LIN {X 0,Y 573.337,Z 321.881,A -85,B 0,C 180,E1 -2340.702,E2 -2340.702} C_VEL
LIN {X 0,Y 573.231,Z 321.897,A -85,B 0,C 180,E1 -2343.514,E2 -2343.514} C_VEL
LIN {X 0,Y 573.289,Z 321.888,A -85,B 0,C 180,E1 -2345.627,E2 -2345.627} C_VEL
LIN {X 0,Y 573.268,Z 321.89,A -85,B 0,C 180,E1 -2347.749,E2 -2347.749} C_VEL
LIN {X 0,Y 573.27,Z 321.892,A -85,B 0,C 180,E1 -2350.596,E2 -2350.596} C_VEL
LIN {X 0,Y 573.267,Z 321.891,A -85,B 0,C 180,E1 -2352.748,E2 -2352.748} C_VEL
LIN {X 0,Y 573.237,Z 321.894,A -85,B 0,C 180,E1 -2354.919,E2 -2354.919} C_VEL
LIN {X 0,Y 573.254,Z 321.892,A -85,B 0,C 180,E1 -2357.111,E2 -2357.111} C_VEL
LIN {X 0,Y 573.125,Z 322.237,A -85,B 0,C 180,E1 -2358.591,E2 -2358.591} C_VEL
LIN {X 0,Y 573.096,Z 326.558,A -85,B 0,C 180,E1 -2361.585,E2 -2361.585} C_VEL
LIN {X 0,Y 573.056,Z 329.759,A -85,B 0,C 180,E1 -2363.872,E2 -2363.872} C_VEL
LIN {X 0,Y 573.047,Z 330.361,A -85,B 0,C 180,E1 -2364.307,E2 -2364.307} C_VEL
LIN {X 0,Y 572.39,Z 331.226,A -85,B 0,C 180,E1 -2364.887,E2 -2364.887} C_VEL
LIN {X 0,Y 569.518,Z 332.787,A -85,B 0,C 180,E1 -2365.825,E2 -2365.825} C_VEL
LIN {X 0,Y 567.073,Z 334.053,A -85,B 0,C 180,E1 -2366.58,E2 -2366.58} C_VEL
LIN {X 0,Y 566.011,Z 334.964,A -85,B 0,C 180,E1 -2367.164,E2 -2367.164} C_VEL
LIN {X 0,Y 565.919,Z 335.251,A -85,B 0,C 180,E1 -2367.362,E2 -2367.362} C_VEL
LIN {X 0,Y 565.876,Z 338.726,A -85,B 0,C 180,E1 -2369.786,E2 -2369.786} C_VEL
LIN {X 0,Y 565.854,Z 342.602,A -85,B 0,C 180,E1 -2372.373,E2 -2372.373} C_VEL
LIN {X 0,Y 565.846,Z 346.578,A -85,B 0,C 180,E1 -2374.94,E2 -2374.94} C_VEL
LIN {X 0,Y 565.825,Z 350.574,A -85,B 0,C 180,E1 -2377.488,E2 -2377.488} C_VEL
LIN {X 0,Y 565.868,Z 354.863,A -85,B 0,C 180,E1 -2380.116,E2 -2380.116} C_VEL
LIN {X 0,Y 566.508,Z 362.319,A -85,B 0,C 180,E1 -2380.33,E2 -2380.33} C_VEL
LIN {X 0,Y 566.389,Z 373.209,A -85,B 0,C 180,E1 -2380.747,E2 -2380.747} C_VEL
LIN {X 0,Y 566.3,Z 382.804,A -85,B 0,C 180,E1 -2381.245,E2 -2381.245} C_VEL
LIN {X 0,Y 566.199,Z 390.332,A -85,B 0,C 180,E1 -2381.733,E2 -2381.733} C_VEL
LIN {X 0,Y 566.136,Z 397.915,A -85,B 0,C 180,E1 -2382.333,E2 -2382.333} C_VEL
LIN {X 0,Y 566.099,Z 405.454,A -85,B 0,C 180,E1 -2383.062,E2 -2383.062} C_VEL
LIN {X 0,Y 566.019,Z 413.662,A -85,B 0,C 180,E1 -2384.052,E2 -2384.052} C_VEL
LIN {X 0,Y 565.982,Z 419.96,A -85,B 0,C 180,E1 -2385.054,E2 -2385.054} C_VEL
LIN {X 0,Y 565.916,Z 424.329,A -85,B 0,C 180,E1 -2385.936,E2 -2385.936} C_VEL
LIN {X 0,Y 565.905,Z 426.671,A -85,B 0,C 180,E1 -2386.499,E2 -2386.499} C_VEL
LIN {X 0,Y 565.894,Z 428.668,A -85,B 0,C 180,E1 -2387.115,E2 -2387.115} C_VEL
LIN {X 0,Y 565.859,Z 431.271,A -85,B 0,C 180,E1 -2388.175,E2 -2388.175} C_VEL
LIN {X 0,Y 565.829,Z 432.675,A -85,B 0,C 180,E1 -2389.257,E2 -2389.257} C_VEL
LIN {X 0,Y 565.843,Z 432.888,A -85,B 0,C 180,E1 -2390.358,E2 -2390.358} C_VEL
LIN {X 0,Y 565.839,Z 431.745,A -85,B 0,C 180,E1 -2391.608,E2 -2391.608} C_VEL
LIN {X 0,Y 565.857,Z 429.634,A -85,B 0,C 180,E1 -2392.642,E2 -2392.642} C_VEL
LIN {X 0,Y 565.92,Z 425.738,A -85,B 0,C 180,E1 -2393.823,E2 -2393.823} C_VEL
LIN {X 0,Y 565.922,Z 421.824,A -85,B 0,C 180,E1 -2394.689,E2 -2394.689} C_VEL
LIN {X 0,Y 565.978,Z 416.587,A -85,B 0,C 180,E1 -2395.597,E2 -2395.597} C_VEL
LIN {X 0,Y 565.996,Z 411.667,A -85,B 0,C 180,E1 -2396.296,E2 -2396.296} C_VEL
LIN {X 0,Y 566.128,Z 404.978,A -85,B 0,C 180,E1 -2397.078,E2 -2397.078} C_VEL
LIN {X 0,Y 566.155,Z 398.125,A -85,B 0,C 180,E1 -2397.738,E2 -2397.738} C_VEL
LIN {X 0,Y 566.21,Z 390.149,A -85,B 0,C 180,E1 -2398.37,E2 -2398.37} C_VEL
LIN {X 0,Y 566.285,Z 380.733,A -85,B 0,C 180,E1 -2398.969,E2 -2398.969} C_VEL
LIN {X 0,Y 566.421,Z 370.239,A -85,B 0,C 180,E1 -2399.472,E2 -2399.472} C_VEL
LIN {X 0,Y 566.469,Z 359.574,A -85,B 0,C 180,E1 -2399.836,E2 -2399.836} C_VEL
LIN {X 0,Y 565.876,Z 354.723,A -85,B 0,C 180,E1 -2399.981,E2 -2399.981} C_VEL
LIN {X 0,Y 565.864,Z 350.509,A -85,B 0,C 180,E1 -2402.642,E2 -2402.642} C_VEL
LIN {X 0,Y 565.92,Z 346.759,A -85,B 0,C 180,E1 -2405.032,E2 -2405.032} C_VEL
LIN {X 0,Y 565.88,Z 341.975,A -85,B 0,C 180,E1 -2408.124,E2 -2408.124} C_VEL
LIN {X 0,Y 565.936,Z 337.526,A -85,B 0,C 180,E1 -2411.162,E2 -2411.162} C_VEL
LIN {X 0,Y 565.952,Z 334.388,A -85,B 0,C 180,E1 -2413.404,E2 -2413.404} C_VEL
LIN {X 0,Y 565.963,Z 330.08,A -85,B 0,C 180,E1 -2416.352,E2 -2416.352} C_VEL
LIN {X 0,Y 566.05,Z 325.919,A -85,B 0,C 180,E1 -2419.266,E2 -2419.266} C_VEL
LIN {X 0,Y 566.057,Z 322.872,A -85,B 0,C 180,E1 -2421.431,E2 -2421.431} C_VEL
LIN {X 0,Y 566.194,Z 322.774,A -85,B 0,C 180,E1 -2423.585,E2 -2423.585} C_VEL
LIN {X 0,Y 566.184,Z 322.773,A -85,B 0,C 180,E1 -2425.728,E2 -2425.728} C_VEL
LIN {X 0,Y 566.267,Z 322.762,A -85,B 0,C 180,E1 -2427.865,E2 -2427.865} C_VEL
LIN {X 0,Y 566.297,Z 322.761,A -85,B 0,C 180,E1 -2430.71,E2 -2430.71} C_VEL
LIN {X 0,Y 566.267,Z 322.762,A -85,B 0,C 180,E1 -2432.845,E2 -2432.845} C_VEL
LIN {X 0,Y 566.253,Z 322.767,A -85,B 0,C 180,E1 -2435.697,E2 -2435.697} C_VEL
LIN {X 0,Y 566.239,Z 322.765,A -85,B 0,C 180,E1 -2438.565,E2 -2438.565} C_VEL
LIN {X 0,Y 566.239,Z 322.766,A -85,B 0,C 180,E1 -2441.453,E2 -2441.453} C_VEL
LIN {X 0,Y 566.221,Z 322.767,A -85,B 0,C 180,E1 -2444.506,E2 -2444.506} C_VEL
LIN {X 0,Y 566.192,Z 322.771,A -85,B 0,C 180,E1 -2447.331,E2 -2447.331} C_VEL
LIN {X 0,Y 566.211,Z 322.771,A -85,B 0,C 180,E1 -2450.336,E2 -2450.336} C_VEL
LIN {X 0,Y 566.177,Z 322.773,A -85,B 0,C 180,E1 -2453.403,E2 -2453.403} C_VEL
LIN {X 0,Y 566.211,Z 322.769,A -85,B 0,C 180,E1 -2455.748,E2 -2455.748} C_VEL
LIN {X 0,Y 566.195,Z 322.77,A -85,B 0,C 180,E1 -2458.203,E2 -2458.203} C_VEL
LIN {X 0,Y 566.182,Z 322.772,A -85,B 0,C 180,E1 -2460.591,E2 -2460.591} C_VEL
LIN {X 0,Y 566.216,Z 322.768,A -85,B 0,C 180,E1 -2463.101,E2 -2463.101} C_VEL
LIN {X 0,Y 566.199,Z 322.771,A -85,B 0,C 180,E1 -2465.688,E2 -2465.688} C_VEL
LIN {X 0,Y 566.202,Z 322.773,A -85,B 0,C 180,E1 -2468.559,E2 -2468.559} C_VEL
LIN {X 0,Y 566.206,Z 322.771,A -85,B 0,C 180,E1 -2471.135,E2 -2471.135} C_VEL
LIN {X 0,Y 566.186,Z 322.771,A -85,B 0,C 180,E1 -2474.035,E2 -2474.035} C_VEL
LIN {X 0,Y 566.19,Z 322.774,A -85,B 0,C 180,E1 -2477.082,E2 -2477.082} C_VEL
LIN {X 0,Y 566.213,Z 322.768,A -85,B 0,C 180,E1 -2479.803,E2 -2479.803} C_VEL
LIN {X 0,Y 566.185,Z 322.772,A -85,B 0,C 180,E1 -2482.599,E2 -2482.599} C_VEL
LIN {X 0,Y 566.208,Z 322.77,A -85,B 0,C 180,E1 -2485.183,E2 -2485.183} C_VEL
LIN {X 0,Y 566.221,Z 322.77,A -85,B 0,C 180,E1 -2487.744,E2 -2487.744} C_VEL
LIN {X 0,Y 566.216,Z 322.771,A -85,B 0,C 180,E1 -2490.323,E2 -2490.323} C_VEL
LIN {X 0,Y 566.207,Z 322.772,A -85,B 0,C 180,E1 -2492.662,E2 -2492.662} C_VEL
LIN {X 0,Y 566.221,Z 322.77,A -85,B 0,C 180,E1 -2495.039,E2 -2495.039} C_VEL
LIN {X 0,Y 566.192,Z 322.773,A -85,B 0,C 180,E1 -2497.37,E2 -2497.37} C_VEL
LIN {X 0,Y 566.206,Z 322.769,A -85,B 0,C 180,E1 -2499.664,E2 -2499.664} C_VEL
LIN {X 0,Y 566.193,Z 322.772,A -85,B 0,C 180,E1 -2502.669,E2 -2502.669} C_VEL
LIN {X 0,Y 566.221,Z 322.767,A -85,B 0,C 180,E1 -2505.627,E2 -2505.627} C_VEL
LIN {X 0,Y 566.221,Z 322.769,A -85,B 0,C 180,E1 -2508.676,E2 -2508.676} C_VEL
LIN {X 0,Y 566.24,Z 322.765,A -85,B 0,C 180,E1 -2511.435,E2 -2511.435} C_VEL
LIN {X 0,Y 566.253,Z 322.765,A -85,B 0,C 180,E1 -2514.302,E2 -2514.302} C_VEL
LIN {X 0,Y 566.277,Z 322.761,A -85,B 0,C 180,E1 -2517.867,E2 -2517.867} C_VEL
LIN {X 0,Y 566.3,Z 322.76,A -85,B 0,C 180,E1 -2520.712,E2 -2520.712} C_VEL
LIN {X 0,Y 566.264,Z 322.763,A -85,B 0,C 180,E1 -2522.846,E2 -2522.846} C_VEL
LIN {X 0,Y 566.251,Z 322.766,A -85,B 0,C 180,E1 -2525.699,E2 -2525.699} C_VEL
LIN {X 0,Y 566.22,Z 322.767,A -85,B 0,C 180,E1 -2528.566,E2 -2528.566} C_VEL
LIN {X 0,Y 566.241,Z 322.767,A -85,B 0,C 180,E1 -2531.455,E2 -2531.455} C_VEL
LIN {X 0,Y 566.225,Z 322.766,A -85,B 0,C 180,E1 -2534.508,E2 -2534.508} C_VEL
LIN {X 0,Y 566.196,Z 322.771,A -85,B 0,C 180,E1 -2537.332,E2 -2537.332} C_VEL
LIN {X 0,Y 566.206,Z 322.77,A -85,B 0,C 180,E1 -2540.338,E2 -2540.338} C_VEL
LIN {X 0,Y 566.182,Z 322.773,A -85,B 0,C 180,E1 -2543.405,E2 -2543.405} C_VEL
LIN {X 0,Y 566.215,Z 322.769,A -85,B 0,C 180,E1 -2545.749,E2 -2545.749} C_VEL
LIN {X 0,Y 566.2,Z 322.77,A -85,B 0,C 180,E1 -2548.204,E2 -2548.204} C_VEL
LIN {X 0,Y 566.179,Z 322.772,A -85,B 0,C 180,E1 -2550.593,E2 -2550.593} C_VEL
LIN {X 0,Y 566.221,Z 322.768,A -85,B 0,C 180,E1 -2553.102,E2 -2553.102} C_VEL
LIN {X 0,Y 566.206,Z 322.771,A -85,B 0,C 180,E1 -2555.689,E2 -2555.689} C_VEL
LIN {X 0,Y 566.21,Z 322.77,A -85,B 0,C 180,E1 -2558.56,E2 -2558.56} C_VEL
LIN {X 0,Y 566.204,Z 322.77,A -85,B 0,C 180,E1 -2561.137,E2 -2561.137} C_VEL
LIN {X 0,Y 566.194,Z 322.771,A -85,B 0,C 180,E1 -2564.036,E2 -2564.036} C_VEL
LIN {X 0,Y 566.199,Z 322.771,A -85,B 0,C 180,E1 -2567.084,E2 -2567.084} C_VEL
LIN {X 0,Y 566.222,Z 322.767,A -85,B 0,C 180,E1 -2569.804,E2 -2569.804} C_VEL
LIN {X 0,Y 566.195,Z 322.771,A -85,B 0,C 180,E1 -2572.6,E2 -2572.6} C_VEL
LIN {X 0,Y 566.218,Z 322.771,A -85,B 0,C 180,E1 -2575.184,E2 -2575.184} C_VEL
LIN {X 0,Y 566.279,Z 322.886,A -85,B 0,C 180,E1 -2576.326,E2 -2576.326} C_VEL
LIN {X 0,Y 566.647,Z 327.07,A -85,B 0,C 180,E1 -2577.771,E2 -2577.771} C_VEL
LIN {X 0,Y 566.5,Z 334.622,A -85,B 0,C 180,E1 -2580.276,E2 -2580.276} C_VEL
LIN {X 0,Y 566.374,Z 343.367,A -85,B 0,C 180,E1 -2583.03,E2 -2583.03} C_VEL
LIN {X 0,Y 566.309,Z 351.29,A -85,B 0,C 180,E1 -2585.435,E2 -2585.435} C_VEL
LIN {X 0,Y 566.255,Z 360.365,A -85,B 0,C 180,E1 -2588.141,E2 -2588.141} C_VEL
LIN {X 0,Y 566.142,Z 370.65,A -85,B 0,C 180,E1 -2591.171,E2 -2591.171} C_VEL
LIN {X 0,Y 566.087,Z 379.591,A -85,B 0,C 180,E1 -2593.78,E2 -2593.78} C_VEL
LIN {X 0,Y 566.031,Z 388.533,A -85,B 0,C 180,E1 -2596.356,E2 -2596.356} C_VEL
LIN {X 0,Y 565.987,Z 397.114,A -85,B 0,C 180,E1 -2598.802,E2 -2598.802} C_VEL
LIN {X 0,Y 565.966,Z 401.306,A -85,B 0,C 180,E1 -2599.989,E2 -2599.989} C_VEL
LIN {X 0,Y 566.514,Z 408.45,A -85,B 0,C 180,E1 -2600.18,E2 -2600.18} C_VEL
LIN {X 0,Y 566.458,Z 416.916,A -85,B 0,C 180,E1 -2600.449,E2 -2600.449} C_VEL
LIN {X 0,Y 566.389,Z 425.418,A -85,B 0,C 180,E1 -2600.808,E2 -2600.808} C_VEL
LIN {X 0,Y 566.316,Z 433.746,A -85,B 0,C 180,E1 -2601.257,E2 -2601.257} C_VEL
LIN {X 0,Y 566.207,Z 441.783,A -85,B 0,C 180,E1 -2601.794,E2 -2601.794} C_VEL
LIN {X 0,Y 566.126,Z 450.442,A -85,B 0,C 180,E1 -2602.511,E2 -2602.511} C_VEL
LIN {X 0,Y 566.069,Z 459.353,A -85,B 0,C 180,E1 -2603.458,E2 -2603.458} C_VEL
LIN {X 0,Y 566.025,Z 465.618,A -85,B 0,C 180,E1 -2604.3,E2 -2604.3} C_VEL
LIN {X 0,Y 565.906,Z 469.993,A -85,B 0,C 180,E1 -2605.014,E2 -2605.014} C_VEL
LIN {X 0,Y 565.943,Z 475.152,A -85,B 0,C 180,E1 -2606.085,E2 -2606.085} C_VEL
LIN {X 0,Y 565.88,Z 478.938,A -85,B 0,C 180,E1 -2607.153,E2 -2607.153} C_VEL
LIN {X 0,Y 565.841,Z 480.684,A -85,B 0,C 180,E1 -2607.866,E2 -2607.866} C_VEL
LIN {X 0,Y 565.844,Z 481.935,A -85,B 0,C 180,E1 -2608.578,E2 -2608.578} C_VEL
LIN {X 0,Y 565.837,Z 482.71,A -85,B 0,C 180,E1 -2609.289,E2 -2609.289} C_VEL
LIN {X 0,Y 565.836,Z 483,A -85,B 0,C 180,E1 -2610.001,E2 -2610.001} C_VEL
LIN {X 0,Y 565.837,Z 482.709,A -85,B 0,C 180,E1 -2610.713,E2 -2610.713} C_VEL
LIN {X 0,Y 565.844,Z 481.933,A -85,B 0,C 180,E1 -2611.424,E2 -2611.424} C_VEL
LIN {X 0,Y 565.841,Z 480.679,A -85,B 0,C 180,E1 -2612.136,E2 -2612.136} C_VEL
LIN {X 0,Y 565.912,Z 477.785,A -85,B 0,C 180,E1 -2613.205,E2 -2613.205} C_VEL
LIN {X 0,Y 565.934,Z 475.144,A -85,B 0,C 180,E1 -2613.917,E2 -2613.917} C_VEL
LIN {X 0,Y 565.906,Z 469.981,A -85,B 0,C 180,E1 -2614.988,E2 -2614.988} C_VEL
LIN {X 0,Y 566.082,Z 463.179,A -85,B 0,C 180,E1 -2616.058,E2 -2616.058} C_VEL
LIN {X 0,Y 566.092,Z 456.174,A -85,B 0,C 180,E1 -2616.907,E2 -2616.907} C_VEL
LIN {X 0,Y 566.149,Z 448.395,A -85,B 0,C 180,E1 -2617.67,E2 -2617.67} C_VEL
LIN {X 0,Y 566.25,Z 440.531,A -85,B 0,C 180,E1 -2618.297,E2 -2618.297} C_VEL
LIN {X 0,Y 566.371,Z 430.715,A -85,B 0,C 180,E1 -2618.924,E2 -2618.924} C_VEL
LIN {X 0,Y 566.436,Z 419.281,A -85,B 0,C 180,E1 -2619.463,E2 -2619.463} C_VEL
LIN {X 0,Y 566.529,Z 409.215,A -85,B 0,C 180,E1 -2619.799,E2 -2619.799} C_VEL
LIN {X 0,Y 566.065,Z 402.339,A -85,B 0,C 180,E1 -2619.977,E2 -2619.977} C_VEL
LIN {X 0,Y 565.967,Z 401.299,A -85,B 0,C 180,E1 -2620.012,E2 -2620.012} C_VEL
LIN {X 0,Y 566.022,Z 392.358,A -85,B 0,C 180,E1 -2622.551,E2 -2622.551} C_VEL
LIN {X 0,Y 566.071,Z 382.139,A -85,B 0,C 180,E1 -2625.483,E2 -2625.483} C_VEL
LIN {X 0,Y 566.15,Z 371.921,A -85,B 0,C 180,E1 -2628.455,E2 -2628.455} C_VEL
LIN {X 0,Y 566.217,Z 362.937,A -85,B 0,C 180,E1 -2631.098,E2 -2631.098} C_VEL
LIN {X 0,Y 566.277,Z 353.823,A -85,B 0,C 180,E1 -2633.789,E2 -2633.789} C_VEL
LIN {X 0,Y 566.357,Z 344.685,A -85,B 0,C 180,E1 -2636.535,E2 -2636.535} C_VEL
LIN {X 0,Y 566.491,Z 335.795,A -85,B 0,C 180,E1 -2639.331,E2 -2639.331} C_VEL
LIN {X 0,Y 566.638,Z 328.27,A -85,B 0,C 180,E1 -2641.812,E2 -2641.812} C_VEL
LIN {X 0,Y 566.387,Z 323.621,A -85,B 0,C 180,E1 -2643.409,E2 -2643.409} C_VEL
LIN {X 0,Y 566.234,Z 322.768,A -85,B 0,C 180,E1 -2643.737,E2 -2643.737} C_VEL
LIN {X 0,Y 566.205,Z 322.77,A -85,B 0,C 180,E1 -2646.57,E2 -2646.57} C_VEL
LIN {X 0,Y 566.217,Z 322.77,A -85,B 0,C 180,E1 -2649.686,E2 -2649.686} C_VEL
LIN {X 0,Y 566.21,Z 322.774,A -85,B 0,C 180,E1 -2652.918,E2 -2652.918} C_VEL
LIN {X 0,Y 566.199,Z 322.772,A -85,B 0,C 180,E1 -2656.049,E2 -2656.049} C_VEL
LIN {X 0,Y 566.209,Z 322.769,A -85,B 0,C 180,E1 -2659.215,E2 -2659.215} C_VEL
LIN {X 0,Y 566.186,Z 322.772,A -85,B 0,C 180,E1 -2661.636,E2 -2661.636} C_VEL
LIN {X 0,Y 566.168,Z 322.775,A -85,B 0,C 180,E1 -2664.308,E2 -2664.308} C_VEL
LIN {X 0,Y 566.207,Z 322.771,A -85,B 0,C 180,E1 -2666.897,E2 -2666.897} C_VEL
LIN {X 0,Y 566.179,Z 322.776,A -85,B 0,C 180,E1 -2669.407,E2 -2669.407} C_VEL
LIN {X 0,Y 566.201,Z 322.773,A -85,B 0,C 180,E1 -2671.856,E2 -2671.856} C_VEL
LIN {X 0,Y 566.216,Z 322.77,A -85,B 0,C 180,E1 -2674.251,E2 -2674.251} C_VEL
LIN {X 0,Y 566.177,Z 322.774,A -85,B 0,C 180,E1 -2676.719,E2 -2676.719} C_VEL
LIN {X 0,Y 566.211,Z 322.769,A -85,B 0,C 180,E1 -2679.662,E2 -2679.662} C_VEL
LIN {X 0,Y 566.204,Z 322.77,A -85,B 0,C 180,E1 -2682.668,E2 -2682.668} C_VEL
LIN {X 0,Y 566.227,Z 322.768,A -85,B 0,C 180,E1 -2685.626,E2 -2685.626} C_VEL
LIN {X 0,Y 566.241,Z 322.765,A -85,B 0,C 180,E1 -2688.675,E2 -2688.675} C_VEL
LIN {X 0,Y 566.209,Z 322.77,A -85,B 0,C 180,E1 -2691.433,E2 -2691.433} C_VEL
LIN {X 0,Y 566.259,Z 322.765,A -85,B 0,C 180,E1 -2694.301,E2 -2694.301} C_VEL
LIN {X 0,Y 566.28,Z 322.762,A -85,B 0,C 180,E1 -2697.866,E2 -2697.866} C_VEL
LIN {X 0,Y 566.308,Z 322.757,A -85,B 0,C 180,E1 -2700.71,E2 -2700.71} C_VEL
LIN {X 0,Y 566.273,Z 322.761,A -85,B 0,C 180,E1 -2702.845,E2 -2702.845} C_VEL
LIN {X 0,Y 566.258,Z 322.764,A -85,B 0,C 180,E1 -2705.698,E2 -2705.698} C_VEL
LIN {X 0,Y 566.223,Z 322.767,A -85,B 0,C 180,E1 -2707.846,E2 -2707.846} C_VEL
LIN {X 0,Y 566.242,Z 322.768,A -85,B 0,C 180,E1 -2710.729,E2 -2710.729} C_VEL
LIN {X 0,Y 566.211,Z 322.771,A -85,B 0,C 180,E1 -2712.909,E2 -2712.909} C_VEL
LIN {X 0,Y 566.201,Z 322.772,A -85,B 0,C 180,E1 -2715.109,E2 -2715.109} C_VEL
LIN {X 0,Y 566.184,Z 322.773,A -85,B 0,C 180,E1 -2717.331,E2 -2717.331} C_VEL
LIN {X 0,Y 566.113,Z 322.784,A -85,B 0,C 180,E1 -2718.08,E2 -2718.08} C_VEL
LIN {X 0,Y 566.063,Z 323.28,A -85,B 0,C 180,E1 -2718.832,E2 -2718.832} C_VEL
LIN {X 0,Y 566.052,Z 326.899,A -85,B 0,C 180,E1 -2721.378,E2 -2721.378} C_VEL
LIN {X 0,Y 565.975,Z 330.828,A -85,B 0,C 180,E1 -2724.19,E2 -2724.19} C_VEL
LIN {X 0,Y 565.972,Z 334.186,A -85,B 0,C 180,E1 -2726.61,E2 -2726.61} C_VEL
LIN {X 0,Y 565.919,Z 335.251,A -85,B 0,C 180,E1 -2727.362,E2 -2727.362} C_VEL
LIN {X 0,Y 565.232,Z 336.148,A -85,B 0,C 180,E1 -2727.95,E2 -2727.95} C_VEL
LIN {X 0,Y 562.353,Z 337.767,A -85,B 0,C 180,E1 -2728.9,E2 -2728.9} C_VEL
LIN {X 0,Y 559.929,Z 339.082,A -85,B 0,C 180,E1 -2729.665,E2 -2729.665} C_VEL
LIN {X 0,Y 558.89,Z 340.031,A -85,B 0,C 180,E1 -2730.256,E2 -2730.256} C_VEL
LIN {X 0,Y 558.805,Z 340.331,A -85,B 0,C 180,E1 -2730.457,E2 -2730.457} C_VEL
LIN {X 0,Y 558.762,Z 343.568,A -85,B 0,C 180,E1 -2732.74,E2 -2732.74} C_VEL
LIN {X 0,Y 558.745,Z 347.513,A -85,B 0,C 180,E1 -2735.351,E2 -2735.351} C_VEL
LIN {X 0,Y 558.732,Z 351.698,A -85,B 0,C 180,E1 -2738.048,E2 -2738.048} C_VEL
LIN {X 0,Y 558.775,Z 354.79,A -85,B 0,C 180,E1 -2739.987,E2 -2739.987} C_VEL
LIN {X 0,Y 559.498,Z 361.692,A -85,B 0,C 180,E1 -2740.189,E2 -2740.189} C_VEL
LIN {X 0,Y 559.414,Z 372.799,A -85,B 0,C 180,E1 -2740.61,E2 -2740.61} C_VEL
LIN {X 0,Y 559.309,Z 381.698,A -85,B 0,C 180,E1 -2741.067,E2 -2741.067} C_VEL
LIN {X 0,Y 559.18,Z 389.687,A -85,B 0,C 180,E1 -2741.581,E2 -2741.581} C_VEL
LIN {X 0,Y 559.132,Z 396.739,A -85,B 0,C 180,E1 -2742.131,E2 -2742.131} C_VEL
LIN {X 0,Y 559.057,Z 404.361,A -85,B 0,C 180,E1 -2742.857,E2 -2742.857} C_VEL
LIN {X 0,Y 558.971,Z 410.72,A -85,B 0,C 180,E1 -2743.594,E2 -2743.594} C_VEL
LIN {X 0,Y 558.903,Z 415.222,A -85,B 0,C 180,E1 -2744.212,E2 -2744.212} C_VEL
LIN {X 0,Y 558.91,Z 420.013,A -85,B 0,C 180,E1 -2745,E2 -2745} C_VEL
LIN {X 0,Y 558.839,Z 423.945,A -85,B 0,C 180,E1 -2745.792,E2 -2745.792} C_VEL
LIN {X 0,Y 558.808,Z 427.909,A -85,B 0,C 180,E1 -2746.839,E2 -2746.839} C_VEL
LIN {X 0,Y 558.769,Z 430.737,A -85,B 0,C 180,E1 -2747.907,E2 -2747.907} C_VEL
LIN {X 0,Y 558.746,Z 432.616,A -85,B 0,C 180,E1 -2749.151,E2 -2749.151} C_VEL
LIN {X 0,Y 558.758,Z 432.993,A -85,B 0,C 180,E1 -2750.106,E2 -2750.106} C_VEL
LIN {X 0,Y 558.731,Z 432.251,A -85,B 0,C 180,E1 -2751.246,E2 -2751.246} C_VEL
LIN {X 0,Y 558.734,Z 431.251,A -85,B 0,C 180,E1 -2751.95,E2 -2751.95} C_VEL
LIN {X 0,Y 558.785,Z 429.141,A -85,B 0,C 180,E1 -2752.863,E2 -2752.863} C_VEL
LIN {X 0,Y 558.845,Z 426.176,A -85,B 0,C 180,E1 -2753.766,E2 -2753.766} C_VEL
LIN {X 0,Y 558.839,Z 421.404,A -85,B 0,C 180,E1 -2754.828,E2 -2754.828} C_VEL
LIN {X 0,Y 558.899,Z 417.435,A -85,B 0,C 180,E1 -2755.537,E2 -2755.537} C_VEL
LIN {X 0,Y 558.949,Z 411.399,A -85,B 0,C 180,E1 -2756.41,E2 -2756.41} C_VEL
LIN {X 0,Y 559.047,Z 404.951,A -85,B 0,C 180,E1 -2757.17,E2 -2757.17} C_VEL
LIN {X 0,Y 559.097,Z 398.37,A -85,B 0,C 180,E1 -2757.814,E2 -2757.814} C_VEL
LIN {X 0,Y 559.166,Z 390.358,A -85,B 0,C 180,E1 -2758.46,E2 -2758.46} C_VEL
LIN {X 0,Y 559.287,Z 380.547,A -85,B 0,C 180,E1 -2759.093,E2 -2759.093} C_VEL
LIN {X 0,Y 559.427,Z 369.369,A -85,B 0,C 180,E1 -2759.624,E2 -2759.624} C_VEL
LIN {X 0,Y 559.443,Z 359.915,A -85,B 0,C 180,E1 -2759.951,E2 -2759.951} C_VEL
LIN {X 0,Y 558.774,Z 354.712,A -85,B 0,C 180,E1 -2760.115,E2 -2760.115} C_VEL
LIN {X 0,Y 558.805,Z 349.825,A -85,B 0,C 180,E1 -2763.244,E2 -2763.244} C_VEL
LIN {X 0,Y 558.814,Z 346.373,A -85,B 0,C 180,E1 -2765.478,E2 -2765.478} C_VEL
LIN {X 0,Y 558.79,Z 342.847,A -85,B 0,C 180,E1 -2767.832,E2 -2767.832} C_VEL
LIN {X 0,Y 558.85,Z 338.459,A -85,B 0,C 180,E1 -2770.914,E2 -2770.914} C_VEL
LIN {X 0,Y 558.873,Z 335.274,A -85,B 0,C 180,E1 -2773.187,E2 -2773.187} C_VEL
LIN {X 0,Y 558.913,Z 330.916,A -85,B 0,C 180,E1 -2776.177,E2 -2776.177} C_VEL
LIN {X 0,Y 558.992,Z 326.76,A -85,B 0,C 180,E1 -2779.129,E2 -2779.129} C_VEL
LIN {X 0,Y 558.999,Z 323.698,A -85,B 0,C 180,E1 -2781.322,E2 -2781.322} C_VEL
LIN {X 0,Y 559.157,Z 323.65,A -85,B 0,C 180,E1 -2783.504,E2 -2783.504} C_VEL
LIN {X 0,Y 559.142,Z 323.65,A -85,B 0,C 180,E1 -2785.674,E2 -2785.674} C_VEL
LIN {X 0,Y 559.239,Z 323.637,A -85,B 0,C 180,E1 -2787.838,E2 -2787.838} C_VEL
LIN {X 0,Y 559.266,Z 323.637,A -85,B 0,C 180,E1 -2790.719,E2 -2790.719} C_VEL
LIN {X 0,Y 559.234,Z 323.638,A -85,B 0,C 180,E1 -2792.88,E2 -2792.88} C_VEL
LIN {X 0,Y 559.222,Z 323.642,A -85,B 0,C 180,E1 -2795.769,E2 -2795.769} C_VEL
LIN {X 0,Y 559.194,Z 323.642,A -85,B 0,C 180,E1 -2798.673,E2 -2798.673} C_VEL
LIN {X 0,Y 559.197,Z 323.644,A -85,B 0,C 180,E1 -2801.6,E2 -2801.6} C_VEL
LIN {X 0,Y 559.186,Z 323.643,A -85,B 0,C 180,E1 -2804.595,E2 -2804.595} C_VEL
LIN {X 0,Y 559.152,Z 323.649,A -85,B 0,C 180,E1 -2807.556,E2 -2807.556} C_VEL
LIN {X 0,Y 559.176,Z 323.645,A -85,B 0,C 180,E1 -2810.603,E2 -2810.603} C_VEL
LIN {X 0,Y 559.134,Z 323.652,A -85,B 0,C 180,E1 -2813.716,E2 -2813.716} C_VEL
LIN {X 0,Y 559.186,Z 323.645,A -85,B 0,C 180,E1 -2816.096,E2 -2816.096} C_VEL
LIN {X 0,Y 559.154,Z 323.649,A -85,B 0,C 180,E1 -2818.529,E2 -2818.529} C_VEL
LIN {X 0,Y 559.144,Z 323.652,A -85,B 0,C 180,E1 -2821.275,E2 -2821.275} C_VEL
LIN {X 0,Y 559.166,Z 323.646,A -85,B 0,C 180,E1 -2823.951,E2 -2823.951} C_VEL
LIN {X 0,Y 559.176,Z 323.645,A -85,B 0,C 180,E1 -2826.451,E2 -2826.451} C_VEL
LIN {X 0,Y 559.164,Z 323.647,A -85,B 0,C 180,E1 -2828.933,E2 -2828.933} C_VEL
LIN {X 0,Y 559.187,Z 323.644,A -85,B 0,C 180,E1 -2831.766,E2 -2831.766} C_VEL
LIN {X 0,Y 559.125,Z 323.653,A -85,B 0,C 180,E1 -2834.739,E2 -2834.739} C_VEL
LIN {X 0,Y 559.149,Z 323.649,A -85,B 0,C 180,E1 -2837.257,E2 -2837.257} C_VEL
LIN {X 0,Y 559.173,Z 323.645,A -85,B 0,C 180,E1 -2840.135,E2 -2840.135} C_VEL
LIN {X 0,Y 559.134,Z 323.653,A -85,B 0,C 180,E1 -2842.892,E2 -2842.892} C_VEL
LIN {X 0,Y 559.149,Z 323.651,A -85,B 0,C 180,E1 -2845.557,E2 -2845.557} C_VEL
LIN {X 0,Y 559.158,Z 323.649,A -85,B 0,C 180,E1 -2848.138,E2 -2848.138} C_VEL
LIN {X 0,Y 559.147,Z 323.65,A -85,B 0,C 180,E1 -2850.648,E2 -2850.648} C_VEL
LIN {X 0,Y 559.158,Z 323.647,A -85,B 0,C 180,E1 -2853.172,E2 -2853.172} C_VEL
LIN {X 0,Y 559.153,Z 323.648,A -85,B 0,C 180,E1 -2855.496,E2 -2855.496} C_VEL
LIN {X 0,Y 559.152,Z 323.649,A -85,B 0,C 180,E1 -2858.448,E2 -2858.448} C_VEL
LIN {X 0,Y 559.16,Z 323.648,A -85,B 0,C 180,E1 -2860.927,E2 -2860.927} C_VEL
LIN {X 0,Y 559.161,Z 323.648,A -85,B 0,C 180,E1 -2863.949,E2 -2863.949} C_VEL
LIN {X 0,Y 559.162,Z 323.65,A -85,B 0,C 180,E1 -2866.185,E2 -2866.185} C_VEL
LIN {X 0,Y 559.192,Z 323.645,A -85,B 0,C 180,E1 -2868.605,E2 -2868.605} C_VEL
LIN {X 0,Y 559.194,Z 323.643,A -85,B 0,C 180,E1 -2871.327,E2 -2871.327} C_VEL
LIN {X 0,Y 559.222,Z 323.64,A -85,B 0,C 180,E1 -2874.231,E2 -2874.231} C_VEL
LIN {X 0,Y 559.248,Z 323.637,A -85,B 0,C 180,E1 -2877.84,E2 -2877.84} C_VEL
LIN {X 0,Y 559.269,Z 323.636,A -85,B 0,C 180,E1 -2880.721,E2 -2880.721} C_VEL
LIN {X 0,Y 559.231,Z 323.64,A -85,B 0,C 180,E1 -2882.882,E2 -2882.882} C_VEL
LIN {X 0,Y 559.22,Z 323.641,A -85,B 0,C 180,E1 -2885.771,E2 -2885.771} C_VEL
LIN {X 0,Y 559.179,Z 323.644,A -85,B 0,C 180,E1 -2888.675,E2 -2888.675} C_VEL
LIN {X 0,Y 559.2,Z 323.646,A -85,B 0,C 180,E1 -2891.601,E2 -2891.601} C_VEL
LIN {X 0,Y 559.19,Z 323.642,A -85,B 0,C 180,E1 -2894.596,E2 -2894.596} C_VEL
LIN {X 0,Y 559.155,Z 323.65,A -85,B 0,C 180,E1 -2897.558,E2 -2897.558} C_VEL
LIN {X 0,Y 559.164,Z 323.648,A -85,B 0,C 180,E1 -2899.838,E2 -2899.838} C_VEL
LIN {X 0,Y 559.134,Z 323.651,A -85,B 0,C 180,E1 -2902.154,E2 -2902.154} C_VEL
LIN {X 0,Y 559.171,Z 323.647,A -85,B 0,C 180,E1 -2905.188,E2 -2905.188} C_VEL
LIN {X 0,Y 559.188,Z 323.644,A -85,B 0,C 180,E1 -2907.712,E2 -2907.712} C_VEL
LIN {X 0,Y 559.158,Z 323.647,A -85,B 0,C 180,E1 -2910.183,E2 -2910.183} C_VEL
LIN {X 0,Y 559.168,Z 323.646,A -85,B 0,C 180,E1 -2912.715,E2 -2912.715} C_VEL
LIN {X 0,Y 559.152,Z 323.648,A -85,B 0,C 180,E1 -2915.323,E2 -2915.323} C_VEL
LIN {X 0,Y 559.129,Z 323.652,A -85,B 0,C 180,E1 -2918.018,E2 -2918.018} C_VEL
LIN {X 0,Y 559.183,Z 323.645,A -85,B 0,C 180,E1 -2921.055,E2 -2921.055} C_VEL
LIN {X 0,Y 559.157,Z 323.647,A -85,B 0,C 180,E1 -2923.733,E2 -2923.733} C_VEL
LIN {X 0,Y 559.162,Z 323.65,A -85,B 0,C 180,E1 -2926.802,E2 -2926.802} C_VEL
LIN {X 0,Y 559.172,Z 323.649,A -85,B 0,C 180,E1 -2929.191,E2 -2929.191} C_VEL
LIN {X 0,Y 559.13,Z 323.651,A -85,B 0,C 180,E1 -2931.984,E2 -2931.984} C_VEL
LIN {X 0,Y 559.156,Z 323.648,A -85,B 0,C 180,E1 -2934.784,E2 -2934.784} C_VEL
LIN {X 0,Y 559.239,Z 323.815,A -85,B 0,C 180,E1 -2936.173,E2 -2936.173} C_VEL
LIN {X 0,Y 559.671,Z 328.303,A -85,B 0,C 180,E1 -2937.746,E2 -2937.746} C_VEL
LIN {X 0,Y 559.509,Z 335.246,A -85,B 0,C 180,E1 -2940.079,E2 -2940.079} C_VEL
LIN {X 0,Y 559.353,Z 343.397,A -85,B 0,C 180,E1 -2942.704,E2 -2942.704} C_VEL
LIN {X 0,Y 559.266,Z 351.32,A -85,B 0,C 180,E1 -2945.144,E2 -2945.144} C_VEL
LIN {X 0,Y 559.206,Z 360.268,A -85,B 0,C 180,E1 -2947.851,E2 -2947.851} C_VEL
LIN {X 0,Y 559.102,Z 369.19,A -85,B 0,C 180,E1 -2950.521,E2 -2950.521} C_VEL
LIN {X 0,Y 559.046,Z 378.314,A -85,B 0,C 180,E1 -2953.194,E2 -2953.194} C_VEL
LIN {X 0,Y 558.982,Z 388.533,A -85,B 0,C 180,E1 -2956.18,E2 -2956.18} C_VEL
LIN {X 0,Y 558.918,Z 398.751,A -85,B 0,C 180,E1 -2959.129,E2 -2959.129} C_VEL
LIN {X 0,Y 558.903,Z 401.306,A -85,B 0,C 180,E1 -2959.862,E2 -2959.862} C_VEL
LIN {X 0,Y 559.537,Z 408.449,A -85,B 0,C 180,E1 -2960.056,E2 -2960.056} C_VEL
LIN {X 0,Y 559.461,Z 416.914,A -85,B 0,C 180,E1 -2960.328,E2 -2960.328} C_VEL
LIN {X 0,Y 559.39,Z 425.415,A -85,B 0,C 180,E1 -2960.692,E2 -2960.692} C_VEL
LIN {X 0,Y 559.296,Z 433.744,A -85,B 0,C 180,E1 -2961.146,E2 -2961.146} C_VEL
LIN {X 0,Y 559.191,Z 441.78,A -85,B 0,C 180,E1 -2961.691,E2 -2961.691} C_VEL
LIN {X 0,Y 559.096,Z 450.443,A -85,B 0,C 180,E1 -2962.417,E2 -2962.417} C_VEL
LIN {X 0,Y 559.002,Z 458.957,A -85,B 0,C 180,E1 -2963.324,E2 -2963.324} C_VEL
LIN {X 0,Y 559.004,Z 464.441,A -85,B 0,C 180,E1 -2964.047,E2 -2964.047} C_VEL
LIN {X 0,Y 558.821,Z 469.994,A -85,B 0,C 180,E1 -2964.95,E2 -2964.95} C_VEL
LIN {X 0,Y 558.858,Z 475.153,A -85,B 0,C 180,E1 -2966.035,E2 -2966.035} C_VEL
LIN {X 0,Y 558.803,Z 478.939,A -85,B 0,C 180,E1 -2967.117,E2 -2967.117} C_VEL
LIN {X 0,Y 558.747,Z 480.685,A -85,B 0,C 180,E1 -2967.838,E2 -2967.838} C_VEL
LIN {X 0,Y 558.744,Z 481.934,A -85,B 0,C 180,E1 -2968.559,E2 -2968.559} C_VEL
LIN {X 0,Y 558.737,Z 482.709,A -85,B 0,C 180,E1 -2969.28,E2 -2969.28} C_VEL
LIN {X 0,Y 558.737,Z 483,A -85,B 0,C 180,E1 -2970.001,E2 -2970.001} C_VEL
LIN {X 0,Y 558.737,Z 482.708,A -85,B 0,C 180,E1 -2970.722,E2 -2970.722} C_VEL
LIN {X 0,Y 558.744,Z 481.931,A -85,B 0,C 180,E1 -2971.442,E2 -2971.442} C_VEL
LIN {X 0,Y 558.747,Z 480.68,A -85,B 0,C 180,E1 -2972.163,E2 -2972.163} C_VEL
LIN {X 0,Y 558.835,Z 477.784,A -85,B 0,C 180,E1 -2973.245,E2 -2973.245} C_VEL
LIN {X 0,Y 558.85,Z 475.145,A -85,B 0,C 180,E1 -2973.967,E2 -2973.967} C_VEL
LIN {X 0,Y 558.822,Z 469.981,A -85,B 0,C 180,E1 -2975.051,E2 -2975.051} C_VEL
LIN {X 0,Y 559.019,Z 463.178,A -85,B 0,C 180,E1 -2976.135,E2 -2976.135} C_VEL
LIN {X 0,Y 559.037,Z 455.736,A -85,B 0,C 180,E1 -2977.041,E2 -2977.041} C_VEL
LIN {X 0,Y 559.123,Z 448.393,A -85,B 0,C 180,E1 -2977.767,E2 -2977.767} C_VEL
LIN {X 0,Y 559.214,Z 440.529,A -85,B 0,C 180,E1 -2978.402,E2 -2978.402} C_VEL
LIN {X 0,Y 559.302,Z 432.213,A -85,B 0,C 180,E1 -2978.947,E2 -2978.947} C_VEL
LIN {X 0,Y 559.437,Z 421.593,A -85,B 0,C 180,E1 -2979.491,E2 -2979.491} C_VEL
LIN {X 0,Y 559.529,Z 410.046,A -85,B 0,C 180,E1 -2979.9,E2 -2979.9} C_VEL
LIN {X 0,Y 559.075,Z 402.986,A -85,B 0,C 180,E1 -2980.091,E2 -2980.091} C_VEL
LIN {X 0,Y 558.904,Z 401.299,A -85,B 0,C 180,E1 -2980.14,E2 -2980.14} C_VEL
LIN {X 0,Y 558.948,Z 392.358,A -85,B 0,C 180,E1 -2982.712,E2 -2982.712} C_VEL
LIN {X 0,Y 559.027,Z 382.139,A -85,B 0,C 180,E1 -2985.683,E2 -2985.683} C_VEL
LIN {X 0,Y 559.104,Z 371.888,A -85,B 0,C 180,E1 -2988.696,E2 -2988.696} C_VEL
LIN {X 0,Y 559.169,Z 362.185,A -85,B 0,C 180,E1 -2991.552,E2 -2991.552} C_VEL
LIN {X 0,Y 559.266,Z 352.386,A -85,B 0,C 180,E1 -2994.501,E2 -2994.501} C_VEL
LIN {X 0,Y 559.35,Z 343.242,A -85,B 0,C 180,E1 -2997.298,E2 -2997.298} C_VEL
LIN {X 0,Y 559.524,Z 334.465,A -85,B 0,C 180,E1 -3000.161,E2 -3000.161} C_VEL
LIN {X 0,Y 559.66,Z 328.224,A -85,B 0,C 180,E1 -3002.256,E2 -3002.256} C_VEL
LIN {X 0,Y 559.266,Z 324.005,A -85,B 0,C 180,E1 -3003.756,E2 -3003.756} C_VEL
LIN {X 0,Y 559.178,Z 323.647,A -85,B 0,C 180,E1 -3003.951,E2 -3003.951} C_VEL
LIN {X 0,Y 559.146,Z 323.652,A -85,B 0,C 180,E1 -3007.109,E2 -3007.109} C_VEL
LIN {X 0,Y 559.163,Z 323.648,A -85,B 0,C 180,E1 -3009.942,E2 -3009.942} C_VEL
LIN {X 0,Y 559.165,Z 323.65,A -85,B 0,C 180,E1 -3012.744,E2 -3012.744} C_VEL
LIN {X 0,Y 559.153,Z 323.649,A -85,B 0,C 180,E1 -3015.762,E2 -3015.762} C_VEL
LIN {X 0,Y 559.168,Z 323.646,A -85,B 0,C 180,E1 -3018.23,E2 -3018.23} C_VEL
LIN {X 0,Y 559.177,Z 323.648,A -85,B 0,C 180,E1 -3021.192,E2 -3021.192} C_VEL
LIN {X 0,Y 559.145,Z 323.65,A -85,B 0,C 180,E1 -3023.789,E2 -3023.789} C_VEL
LIN {X 0,Y 559.153,Z 323.648,A -85,B 0,C 180,E1 -3026.424,E2 -3026.424} C_VEL
LIN {X 0,Y 559.157,Z 323.648,A -85,B 0,C 180,E1 -3028.98,E2 -3028.98} C_VEL
LIN {X 0,Y 559.152,Z 323.65,A -85,B 0,C 180,E1 -3031.623,E2 -3031.623} C_VEL
LIN {X 0,Y 559.184,Z 323.646,A -85,B 0,C 180,E1 -3033.903,E2 -3033.903} C_VEL
LIN {X 0,Y 559.146,Z 323.651,A -85,B 0,C 180,E1 -3036.571,E2 -3036.571} C_VEL
LIN {X 0,Y 559.181,Z 323.644,A -85,B 0,C 180,E1 -3039.395,E2 -3039.395} C_VEL
LIN {X 0,Y 559.143,Z 323.649,A -85,B 0,C 180,E1 -3041.685,E2 -3041.685} C_VEL
LIN {X 0,Y 559.167,Z 323.647,A -85,B 0,C 180,E1 -3043.947,E2 -3043.947} C_VEL
LIN {X 0,Y 559.171,Z 323.647,A -85,B 0,C 180,E1 -3046.184,E2 -3046.184} C_VEL
LIN {X 0,Y 559.212,Z 323.641,A -85,B 0,C 180,E1 -3048.604,E2 -3048.604} C_VEL
LIN {X 0,Y 559.201,Z 323.643,A -85,B 0,C 180,E1 -3052.053,E2 -3052.053} C_VEL
LIN {X 0,Y 559.258,Z 323.635,A -85,B 0,C 180,E1 -3054.953,E2 -3054.953} C_VEL
LIN {X 0,Y 559.251,Z 323.637,A -85,B 0,C 180,E1 -3057.839,E2 -3057.839} C_VEL
LIN {X 0,Y 559.278,Z 323.632,A -85,B 0,C 180,E1 -3060.719,E2 -3060.719} C_VEL
LIN {X 0,Y 559.24,Z 323.637,A -85,B 0,C 180,E1 -3062.881,E2 -3062.881} C_VEL
LIN {X 0,Y 559.229,Z 323.64,A -85,B 0,C 180,E1 -3065.769,E2 -3065.769} C_VEL
LIN {X 0,Y 559.167,Z 323.647,A -85,B 0,C 180,E1 -3068.674,E2 -3068.674} C_VEL
LIN {X 0,Y 559.209,Z 323.642,A -85,B 0,C 180,E1 -3071.599,E2 -3071.599} C_VEL
LIN {X 0,Y 559.203,Z 323.643,A -85,B 0,C 180,E1 -3074.595,E2 -3074.595} C_VEL
LIN {X 0,Y 559.114,Z 323.655,A -85,B 0,C 180,E1 -3077.557,E2 -3077.557} C_VEL
LIN {X 0,Y 559.047,Z 323.665,A -85,B 0,C 180,E1 -3078.317,E2 -3078.317} C_VEL
LIN {X 0,Y 558.988,Z 324.857,A -85,B 0,C 180,E1 -3079.445,E2 -3079.445} C_VEL
LIN {X 0,Y 558.962,Z 328.665,A -85,B 0,C 180,E1 -3082.159,E2 -3082.159} C_VEL
LIN {X 0,Y 558.913,Z 332.73,A -85,B 0,C 180,E1 -3085.127,E2 -3085.127} C_VEL
LIN {X 0,Y 558.836,Z 336.373,A -85,B 0,C 180,E1 -3087.73,E2 -3087.73} C_VEL
LIN {X 0,Y 558.805,Z 340.331,A -85,B 0,C 180,E1 -3090.457,E2 -3090.457} C_VEL
LIN {X 0,Y 558.133,Z 341.262,A -85,B 0,C 180,E1 -3091.051,E2 -3091.051} C_VEL
LIN {X 0,Y 555.254,Z 342.861,A -85,B 0,C 180,E1 -3092.013,E2 -3092.013} C_VEL
LIN {X 0,Y 552.815,Z 344.147,A -85,B 0,C 180,E1 -3092.788,E2 -3092.788} C_VEL
LIN {X 0,Y 551.761,Z 345.07,A -85,B 0,C 180,E1 -3093.387,E2 -3093.387} C_VEL
LIN {X 0,Y 551.672,Z 345.362,A -85,B 0,C 180,E1 -3093.59,E2 -3093.59} C_VEL
LIN {X 0,Y 551.662,Z 348.608,A -85,B 0,C 180,E1 -3095.874,E2 -3095.874} C_VEL
LIN {X 0,Y 551.639,Z 353.405,A -85,B 0,C 180,E1 -3098.999,E2 -3098.999} C_VEL
LIN {X 0,Y 551.671,Z 354.715,A -85,B 0,C 180,E1 -3099.846,E2 -3099.846} C_VEL
LIN {X 0,Y 552.52,Z 363.25,A -85,B 0,C 180,E1 -3100.112,E2 -3100.112} C_VEL
LIN {X 0,Y 552.396,Z 373.304,A -85,B 0,C 180,E1 -3100.514,E2 -3100.514} C_VEL
LIN {X 0,Y 552.267,Z 382.592,A -85,B 0,C 180,E1 -3101.007,E2 -3101.007} C_VEL
LIN {X 0,Y 552.119,Z 390.95,A -85,B 0,C 180,E1 -3101.566,E2 -3101.566} C_VEL
LIN {X 0,Y 552.049,Z 398.306,A -85,B 0,C 180,E1 -3102.171,E2 -3102.171} C_VEL
LIN {X 0,Y 551.981,Z 405.929,A -85,B 0,C 180,E1 -3102.934,E2 -3102.934} C_VEL
LIN {X 0,Y 551.898,Z 412.13,A -85,B 0,C 180,E1 -3103.694,E2 -3103.694} C_VEL
LIN {X 0,Y 551.817,Z 418.881,A -85,B 0,C 180,E1 -3104.72,E2 -3104.72} C_VEL
LIN {X 0,Y 551.76,Z 424.131,A -85,B 0,C 180,E1 -3105.782,E2 -3105.782} C_VEL
LIN {X 0,Y 551.735,Z 427.147,A -85,B 0,C 180,E1 -3106.556,E2 -3106.556} C_VEL
LIN {X 0,Y 551.684,Z 430.191,A -85,B 0,C 180,E1 -3107.634,E2 -3107.634} C_VEL
LIN {X 0,Y 551.662,Z 432.123,A -85,B 0,C 180,E1 -3108.731,E2 -3108.731} C_VEL
LIN {X 0,Y 551.642,Z 432.942,A -85,B 0,C 180,E1 -3109.853,E2 -3109.853} C_VEL
LIN {X 0,Y 551.637,Z 432.575,A -85,B 0,C 180,E1 -3110.999,E2 -3110.999} C_VEL
LIN {X 0,Y 551.662,Z 430.537,A -85,B 0,C 180,E1 -3112.301,E2 -3112.301} C_VEL
LIN {X 0,Y 551.705,Z 428.134,A -85,B 0,C 180,E1 -3113.221,E2 -3113.221} C_VEL
LIN {X 0,Y 551.737,Z 424.871,A -85,B 0,C 180,E1 -3114.129,E2 -3114.129} C_VEL
LIN {X 0,Y 551.765,Z 420.684,A -85,B 0,C 180,E1 -3115.027,E2 -3115.027} C_VEL
LIN {X 0,Y 551.802,Z 415.467,A -85,B 0,C 180,E1 -3115.916,E2 -3115.916} C_VEL
LIN {X 0,Y 551.932,Z 409.002,A -85,B 0,C 180,E1 -3116.801,E2 -3116.801} C_VEL
LIN {X 0,Y 552.036,Z 399.811,A -85,B 0,C 180,E1 -3117.783,E2 -3117.783} C_VEL
LIN {X 0,Y 552.122,Z 392.01,A -85,B 0,C 180,E1 -3118.444,E2 -3118.444} C_VEL
LIN {X 0,Y 552.199,Z 384.426,A -85,B 0,C 180,E1 -3118.971,E2 -3118.971} C_VEL
LIN {X 0,Y 552.289,Z 376.876,A -85,B 0,C 180,E1 -3119.401,E2 -3119.401} C_VEL
LIN {X 0,Y 552.431,Z 368.847,A -85,B 0,C 180,E1 -3119.767,E2 -3119.767} C_VEL
LIN {X 0,Y 552.431,Z 360.438,A -85,B 0,C 180,E1 -3120.063,E2 -3120.063} C_VEL
LIN {X 0,Y 551.681,Z 354.709,A -85,B 0,C 180,E1 -3120.248,E2 -3120.248} C_VEL
LIN {X 0,Y 551.7,Z 350.331,A -85,B 0,C 180,E1 -3123.087,E2 -3123.087} C_VEL
LIN {X 0,Y 551.713,Z 346.084,A -85,B 0,C 180,E1 -3125.943,E2 -3125.943} C_VEL
LIN {X 0,Y 551.715,Z 342.542,A -85,B 0,C 180,E1 -3128.417,E2 -3128.417} C_VEL
LIN {X 0,Y 551.788,Z 339.391,A -85,B 0,C 180,E1 -3130.66,E2 -3130.66} C_VEL
LIN {X 0,Y 551.809,Z 336.11,A -85,B 0,C 180,E1 -3132.965,E2 -3132.965} C_VEL
LIN {X 0,Y 551.828,Z 331.763,A -85,B 0,C 180,E1 -3135.996,E2 -3135.996} C_VEL
LIN {X 0,Y 551.941,Z 327.593,A -85,B 0,C 180,E1 -3138.988,E2 -3138.988} C_VEL
LIN {X 0,Y 551.95,Z 324.548,A -85,B 0,C 180,E1 -3141.21,E2 -3141.21} C_VEL
LIN {X 0,Y 552.124,Z 324.525,A -85,B 0,C 180,E1 -3143.421,E2 -3143.421} C_VEL
LIN {X 0,Y 552.222,Z 324.513,A -85,B 0,C 180,E1 -3144.888,E2 -3144.888} C_VEL
LIN {X 0,Y 552.211,Z 324.513,A -85,B 0,C 180,E1 -3147.811,E2 -3147.811} C_VEL
LIN {X 0,Y 552.236,Z 324.512,A -85,B 0,C 180,E1 -3150.728,E2 -3150.728} C_VEL
LIN {X 0,Y 552.2,Z 324.515,A -85,B 0,C 180,E1 -3152.917,E2 -3152.917} C_VEL
LIN {X 0,Y 552.192,Z 324.517,A -85,B 0,C 180,E1 -3155.843,E2 -3155.843} C_VEL
LIN {X 0,Y 552.162,Z 324.518,A -85,B 0,C 180,E1 -3158.785,E2 -3158.785} C_VEL
LIN {X 0,Y 552.153,Z 324.523,A -85,B 0,C 180,E1 -3161.75,E2 -3161.75} C_VEL
LIN {X 0,Y 552.124,Z 324.523,A -85,B 0,C 180,E1 -3164.748,E2 -3164.748} C_VEL
LIN {X 0,Y 552.103,Z 324.529,A -85,B 0,C 180,E1 -3167.788,E2 -3167.788} C_VEL
LIN {X 0,Y 552.123,Z 324.526,A -85,B 0,C 180,E1 -3170.1,E2 -3170.1} C_VEL
LIN {X 0,Y 552.084,Z 324.53,A -85,B 0,C 180,E1 -3172.45,E2 -3172.45} C_VEL
LIN {X 0,Y 552.143,Z 324.523,A -85,B 0,C 180,E1 -3175.35,E2 -3175.35} C_VEL
LIN {X 0,Y 552.114,Z 324.524,A -85,B 0,C 180,E1 -3178.097,E2 -3178.097} C_VEL
LIN {X 0,Y 552.102,Z 324.526,A -85,B 0,C 180,E1 -3180.608,E2 -3180.608} C_VEL
LIN {X 0,Y 552.116,Z 324.525,A -85,B 0,C 180,E1 -3183.184,E2 -3183.184} C_VEL
LIN {X 0,Y 552.1,Z 324.528,A -85,B 0,C 180,E1 -3185.841,E2 -3185.841} C_VEL
LIN {X 0,Y 552.112,Z 324.525,A -85,B 0,C 180,E1 -3189.062,E2 -3189.062} C_VEL
LIN {X 0,Y 552.157,Z 324.519,A -85,B 0,C 180,E1 -3191.441,E2 -3191.441} C_VEL
LIN {X 0,Y 552.081,Z 324.531,A -85,B 0,C 180,E1 -3194.532,E2 -3194.532} C_VEL
LIN {X 0,Y 552.115,Z 324.524,A -85,B 0,C 180,E1 -3197.584,E2 -3197.584} C_VEL
LIN {X 0,Y 552.121,Z 324.525,A -85,B 0,C 180,E1 -3200.474,E2 -3200.474} C_VEL
LIN {X 0,Y 552.108,Z 324.526,A -85,B 0,C 180,E1 -3203.315,E2 -3203.315} C_VEL
LIN {X 0,Y 552.127,Z 324.523,A -85,B 0,C 180,E1 -3205.94,E2 -3205.94} C_VEL
LIN {X 0,Y 552.103,Z 324.526,A -85,B 0,C 180,E1 -3208.541,E2 -3208.541} C_VEL
LIN {X 0,Y 552.114,Z 324.527,A -85,B 0,C 180,E1 -3211.437,E2 -3211.437} C_VEL
LIN {X 0,Y 552.116,Z 324.525,A -85,B 0,C 180,E1 -3214.356,E2 -3214.356} C_VEL
LIN {X 0,Y 552.128,Z 324.523,A -85,B 0,C 180,E1 -3216.76,E2 -3216.76} C_VEL
LIN {X 0,Y 552.114,Z 324.525,A -85,B 0,C 180,E1 -3219.121,E2 -3219.121} C_VEL
LIN {X 0,Y 552.12,Z 324.525,A -85,B 0,C 180,E1 -3221.445,E2 -3221.445} C_VEL
LIN {X 0,Y 552.11,Z 324.528,A -85,B 0,C 180,E1 -3223.738,E2 -3223.738} C_VEL
LIN {X 0,Y 552.124,Z 324.526,A -85,B 0,C 180,E1 -3226.005,E2 -3226.005} C_VEL
LIN {X 0,Y 552.149,Z 324.52,A -85,B 0,C 180,E1 -3228.994,E2 -3228.994} C_VEL
LIN {X 0,Y 552.153,Z 324.521,A -85,B 0,C 180,E1 -3231.952,E2 -3231.952} C_VEL
LIN {X 0,Y 552.222,Z 324.512,A -85,B 0,C 180,E1 -3234.89,E2 -3234.89} C_VEL
LIN {X 0,Y 552.219,Z 324.512,A -85,B 0,C 180,E1 -3237.813,E2 -3237.813} C_VEL
LIN {X 0,Y 552.239,Z 324.511,A -85,B 0,C 180,E1 -3240.73,E2 -3240.73} C_VEL
LIN {X 0,Y 552.198,Z 324.516,A -85,B 0,C 180,E1 -3242.919,E2 -3242.919} C_VEL
LIN {X 0,Y 552.19,Z 324.516,A -85,B 0,C 180,E1 -3245.845,E2 -3245.845} C_VEL
LIN {X 0,Y 552.15,Z 324.52,A -85,B 0,C 180,E1 -3248.786,E2 -3248.786} C_VEL
LIN {X 0,Y 552.155,Z 324.522,A -85,B 0,C 180,E1 -3251.751,E2 -3251.751} C_VEL
LIN {X 0,Y 552.127,Z 324.522,A -85,B 0,C 180,E1 -3254.749,E2 -3254.749} C_VEL
LIN {X 0,Y 552.106,Z 324.528,A -85,B 0,C 180,E1 -3257.789,E2 -3257.789} C_VEL
LIN {X 0,Y 552.122,Z 324.526,A -85,B 0,C 180,E1 -3260.102,E2 -3260.102} C_VEL
LIN {X 0,Y 552.088,Z 324.53,A -85,B 0,C 180,E1 -3262.452,E2 -3262.452} C_VEL
LIN {X 0,Y 552.148,Z 324.521,A -85,B 0,C 180,E1 -3265.352,E2 -3265.352} C_VEL
LIN {X 0,Y 552.12,Z 324.524,A -85,B 0,C 180,E1 -3268.098,E2 -3268.098} C_VEL
LIN {X 0,Y 552.102,Z 324.526,A -85,B 0,C 180,E1 -3270.61,E2 -3270.61} C_VEL
LIN {X 0,Y 552.122,Z 324.525,A -85,B 0,C 180,E1 -3273.186,E2 -3273.186} C_VEL
LIN {X 0,Y 552.107,Z 324.528,A -85,B 0,C 180,E1 -3275.842,E2 -3275.842} C_VEL
LIN {X 0,Y 552.119,Z 324.525,A -85,B 0,C 180,E1 -3279.063,E2 -3279.063} C_VEL
LIN {X 0,Y 552.133,Z 324.522,A -85,B 0,C 180,E1 -3281.445,E2 -3281.445} C_VEL
LIN {X 0,Y 552.091,Z 324.53,A -85,B 0,C 180,E1 -3284.533,E2 -3284.533} C_VEL
LIN {X 0,Y 552.125,Z 324.523,A -85,B 0,C 180,E1 -3287.586,E2 -3287.586} C_VEL
LIN {X 0,Y 552.129,Z 324.526,A -85,B 0,C 180,E1 -3290.474,E2 -3290.474} C_VEL
LIN {X 0,Y 552.111,Z 324.525,A -85,B 0,C 180,E1 -3293.317,E2 -3293.317} C_VEL
LIN {X 0,Y 552.196,Z 324.546,A -85,B 0,C 180,E1 -3295.945,E2 -3295.945} C_VEL
LIN {X 0,Y 552.709,Z 329.53,A -85,B 0,C 180,E1 -3297.722,E2 -3297.722} C_VEL
LIN {X 0,Y 552.483,Z 338.253,A -85,B 0,C 180,E1 -3300.677,E2 -3300.677} C_VEL
LIN {X 0,Y 552.351,Z 345.288,A -85,B 0,C 180,E1 -3302.957,E2 -3302.957} C_VEL
LIN {X 0,Y 552.241,Z 353.689,A -85,B 0,C 180,E1 -3305.57,E2 -3305.57} C_VEL
LIN {X 0,Y 552.124,Z 362.686,A -85,B 0,C 180,E1 -3308.339,E2 -3308.339} C_VEL
LIN {X 0,Y 552.041,Z 371.667,A -85,B 0,C 180,E1 -3311.057,E2 -3311.057} C_VEL
LIN {X 0,Y 551.957,Z 380.847,A -85,B 0,C 180,E1 -3313.734,E2 -3313.734} C_VEL
LIN {X 0,Y 551.905,Z 389.81,A -85,B 0,C 180,E1 -3316.375,E2 -3316.375} C_VEL
LIN {X 0,Y 551.855,Z 398.751,A -85,B 0,C 180,E1 -3318.988,E2 -3318.988} C_VEL
LIN {X 0,Y 551.839,Z 401.306,A -85,B 0,C 180,E1 -3319.73,E2 -3319.73} C_VEL
LIN {X 0,Y 552.544,Z 410.111,A -85,B 0,C 180,E1 -3319.975,E2 -3319.975} C_VEL
LIN {X 0,Y 552.435,Z 421.632,A -85,B 0,C 180,E1 -3320.389,E2 -3320.389} C_VEL
LIN {X 0,Y 552.274,Z 432.241,A -85,B 0,C 180,E1 -3320.94,E2 -3320.94} C_VEL
LIN {X 0,Y 552.189,Z 440.549,A -85,B 0,C 180,E1 -3321.492,E2 -3321.492} C_VEL
LIN {X 0,Y 552.076,Z 448.407,A -85,B 0,C 180,E1 -3322.135,E2 -3322.135} C_VEL
LIN {X 0,Y 551.99,Z 455.92,A -85,B 0,C 180,E1 -3322.888,E2 -3322.888} C_VEL
LIN {X 0,Y 551.956,Z 463.431,A -85,B 0,C 180,E1 -3323.82,E2 -3323.82} C_VEL
LIN {X 0,Y 551.743,Z 469.994,A -85,B 0,C 180,E1 -3324.885,E2 -3324.885} C_VEL
LIN {X 0,Y 551.778,Z 475.153,A -85,B 0,C 180,E1 -3325.984,E2 -3325.984} C_VEL
LIN {X 0,Y 551.729,Z 478.939,A -85,B 0,C 180,E1 -3327.08,E2 -3327.08} C_VEL
LIN {X 0,Y 551.657,Z 480.684,A -85,B 0,C 180,E1 -3327.811,E2 -3327.811} C_VEL
LIN {X 0,Y 551.644,Z 481.933,A -85,B 0,C 180,E1 -3328.541,E2 -3328.541} C_VEL
LIN {X 0,Y 551.638,Z 482.708,A -85,B 0,C 180,E1 -3329.271,E2 -3329.271} C_VEL
LIN {X 0,Y 551.637,Z 483,A -85,B 0,C 180,E1 -3330.001,E2 -3330.001} C_VEL
LIN {X 0,Y 551.638,Z 482.707,A -85,B 0,C 180,E1 -3330.731,E2 -3330.731} C_VEL
LIN {X 0,Y 551.644,Z 481.93,A -85,B 0,C 180,E1 -3331.461,E2 -3331.461} C_VEL
LIN {X 0,Y 551.658,Z 480.679,A -85,B 0,C 180,E1 -3332.191,E2 -3332.191} C_VEL
LIN {X 0,Y 551.76,Z 477.784,A -85,B 0,C 180,E1 -3333.287,E2 -3333.287} C_VEL
LIN {X 0,Y 551.772,Z 475.145,A -85,B 0,C 180,E1 -3334.018,E2 -3334.018} C_VEL
LIN {X 0,Y 551.743,Z 469.981,A -85,B 0,C 180,E1 -3335.116,E2 -3335.116} C_VEL
LIN {X 0,Y 551.957,Z 463.398,A -85,B 0,C 180,E1 -3336.184,E2 -3336.184} C_VEL
LIN {X 0,Y 551.995,Z 455.735,A -85,B 0,C 180,E1 -3337.132,E2 -3337.132} C_VEL
LIN {X 0,Y 552.078,Z 448.391,A -85,B 0,C 180,E1 -3337.866,E2 -3337.866} C_VEL
LIN {X 0,Y 552.19,Z 440.526,A -85,B 0,C 180,E1 -3338.509,E2 -3338.509} C_VEL
LIN {X 0,Y 552.279,Z 432.211,A -85,B 0,C 180,E1 -3339.061,E2 -3339.061} C_VEL
LIN {X 0,Y 552.449,Z 421.592,A -85,B 0,C 180,E1 -3339.613,E2 -3339.613} C_VEL
LIN {X 0,Y 552.559,Z 410.045,A -85,B 0,C 180,E1 -3340.027,E2 -3340.027} C_VEL
LIN {X 0,Y 552.017,Z 402.985,A -85,B 0,C 180,E1 -3340.222,E2 -3340.222} C_VEL
LIN {X 0,Y 551.839,Z 401.299,A -85,B 0,C 180,E1 -3340.272,E2 -3340.272} C_VEL
LIN {X 0,Y 551.86,Z 391.081,A -85,B 0,C 180,E1 -3343.253,E2 -3343.253} C_VEL
LIN {X 0,Y 551.95,Z 382.139,A -85,B 0,C 180,E1 -3345.889,E2 -3345.889} C_VEL
LIN {X 0,Y 552.022,Z 372.931,A -85,B 0,C 180,E1 -3348.56,E2 -3348.56} C_VEL
LIN {X 0,Y 552.096,Z 363.838,A -85,B 0,C 180,E1 -3351.273,E2 -3351.273} C_VEL
LIN {X 0,Y 552.228,Z 353.544,A -85,B 0,C 180,E1 -3354.433,E2 -3354.433} C_VEL
LIN {X 0,Y 552.307,Z 345.151,A -85,B 0,C 180,E1 -3357.034,E2 -3357.034} C_VEL
LIN {X 0,Y 552.488,Z 336.89,A -85,B 0,C 180,E1 -3359.743,E2 -3359.743} C_VEL
LIN {X 0,Y 552.68,Z 329.421,A -85,B 0,C 180,E1 -3362.282,E2 -3362.282} C_VEL
LIN {X 0,Y 552.343,Z 325.755,A -85,B 0,C 180,E1 -3363.608,E2 -3363.608} C_VEL
LIN {X 0,Y 552.137,Z 324.525,A -85,B 0,C 180,E1 -3364.104,E2 -3364.104} C_VEL
LIN {X 0,Y 552.111,Z 324.527,A -85,B 0,C 180,E1 -3366.747,E2 -3366.747} C_VEL
LIN {X 0,Y 552.132,Z 324.526,A -85,B 0,C 180,E1 -3369.528,E2 -3369.528} C_VEL
LIN {X 0,Y 552.136,Z 324.524,A -85,B 0,C 180,E1 -3372.426,E2 -3372.426} C_VEL
LIN {X 0,Y 552.097,Z 324.529,A -85,B 0,C 180,E1 -3375.562,E2 -3375.562} C_VEL
LIN {X 0,Y 552.126,Z 324.525,A -85,B 0,C 180,E1 -3378.554,E2 -3378.554} C_VEL
LIN {X 0,Y 552.12,Z 324.525,A -85,B 0,C 180,E1 -3381.411,E2 -3381.411} C_VEL
LIN {X 0,Y 552.091,Z 324.528,A -85,B 0,C 180,E1 -3384.156,E2 -3384.156} C_VEL
LIN {X 0,Y 552.112,Z 324.526,A -85,B 0,C 180,E1 -3386.814,E2 -3386.814} C_VEL
LIN {X 0,Y 552.104,Z 324.529,A -85,B 0,C 180,E1 -3389.39,E2 -3389.39} C_VEL
LIN {X 0,Y 552.099,Z 324.529,A -85,B 0,C 180,E1 -3391.901,E2 -3391.901} C_VEL
LIN {X 0,Y 552.162,Z 324.519,A -85,B 0,C 180,E1 -3394.65,E2 -3394.65} C_VEL
LIN {X 0,Y 552.098,Z 324.529,A -85,B 0,C 180,E1 -3397.549,E2 -3397.549} C_VEL
LIN {X 0,Y 552.151,Z 324.521,A -85,B 0,C 180,E1 -3400.375,E2 -3400.375} C_VEL
LIN {X 0,Y 552.14,Z 324.521,A -85,B 0,C 180,E1 -3402.976,E2 -3402.976} C_VEL
LIN {X 0,Y 552.137,Z 324.524,A -85,B 0,C 180,E1 -3406.004,E2 -3406.004} C_VEL
LIN {X 0,Y 552.167,Z 324.518,A -85,B 0,C 180,E1 -3408.993,E2 -3408.993} C_VEL
LIN {X 0,Y 552.155,Z 324.522,A -85,B 0,C 180,E1 -3411.951,E2 -3411.951} C_VEL
LIN {X 0,Y 552.232,Z 324.51,A -85,B 0,C 180,E1 -3414.888,E2 -3414.888} C_VEL
LIN {X 0,Y 552.223,Z 324.513,A -85,B 0,C 180,E1 -3417.811,E2 -3417.811} C_VEL
LIN {X 0,Y 552.248,Z 324.508,A -85,B 0,C 180,E1 -3420.728,E2 -3420.728} C_VEL
LIN {X 0,Y 552.207,Z 324.513,A -85,B 0,C 180,E1 -3422.917,E2 -3422.917} C_VEL
LIN {X 0,Y 552.2,Z 324.516,A -85,B 0,C 180,E1 -3425.843,E2 -3425.843} C_VEL
LIN {X 0,Y 552.14,Z 324.522,A -85,B 0,C 180,E1 -3428.785,E2 -3428.785} C_VEL
LIN {X 0,Y 552.166,Z 324.521,A -85,B 0,C 180,E1 -3431.75,E2 -3431.75} C_VEL
LIN {X 0,Y 552.14,Z 324.523,A -85,B 0,C 180,E1 -3434.747,E2 -3434.747} C_VEL
LIN {X 0,Y 552.106,Z 324.527,A -85,B 0,C 180,E1 -3437.309,E2 -3437.309} C_VEL
LIN {X 0,Y 551.959,Z 324.547,A -85,B 0,C 180,E1 -3438.56,E2 -3438.56} C_VEL
LIN {X 0,Y 551.895,Z 327.551,A -85,B 0,C 180,E1 -3440.888,E2 -3440.888} C_VEL
LIN {X 0,Y 551.87,Z 331.232,A -85,B 0,C 180,E1 -3443.52,E2 -3443.52} C_VEL
LIN {X 0,Y 551.824,Z 335.269,A -85,B 0,C 180,E1 -3446.471,E2 -3446.471} C_VEL
LIN {X 0,Y 551.75,Z 338.772,A -85,B 0,C 180,E1 -3448.948,E2 -3448.948} C_VEL
LIN {X 0,Y 551.721,Z 342.428,A -85,B 0,C 180,E1 -3451.483,E2 -3451.483} C_VEL
LIN {X 0,Y 551.672,Z 345.362,A -85,B 0,C 180,E1 -3453.59,E2 -3453.59} C_VEL
LIN {X 0,Y 550.987,Z 346.267,A -85,B 0,C 180,E1 -3454.193,E2 -3454.193} C_VEL
LIN {X 0,Y 548.097,Z 347.879,A -85,B 0,C 180,E1 -3455.168,E2 -3455.168} C_VEL
LIN {X 0,Y 545.669,Z 349.182,A -85,B 0,C 180,E1 -3455.953,E2 -3455.953} C_VEL
LIN {X 0,Y 544.639,Z 350.125,A -85,B 0,C 180,E1 -3456.56,E2 -3456.56} C_VEL
LIN {X 0,Y 544.561,Z 350.424,A -85,B 0,C 180,E1 -3456.766,E2 -3456.766} C_VEL
LIN {X 0,Y 544.58,Z 354.723,A -85,B 0,C 180,E1 -3459.717,E2 -3459.717} C_VEL
LIN {X 0,Y 545.537,Z 363.115,A -85,B 0,C 180,E1 -3459.979,E2 -3459.979} C_VEL
LIN {X 0,Y 545.369,Z 374.402,A -85,B 0,C 180,E1 -3460.445,E2 -3460.445} C_VEL
LIN {X 0,Y 545.25,Z 383.341,A -85,B 0,C 180,E1 -3460.936,E2 -3460.936} C_VEL
LIN {X 0,Y 545.079,Z 391.829,A -85,B 0,C 180,E1 -3461.523,E2 -3461.523} C_VEL
LIN {X 0,Y 544.988,Z 400.313,A -85,B 0,C 180,E1 -3462.251,E2 -3462.251} C_VEL
LIN {X 0,Y 544.874,Z 408.42,A -85,B 0,C 180,E1 -3463.125,E2 -3463.125} C_VEL
LIN {X 0,Y 544.783,Z 414.375,A -85,B 0,C 180,E1 -3463.926,E2 -3463.926} C_VEL
LIN {X 0,Y 544.732,Z 419.644,A -85,B 0,C 180,E1 -3464.797,E2 -3464.797} C_VEL
LIN {X 0,Y 544.683,Z 424.56,A -85,B 0,C 180,E1 -3465.832,E2 -3465.832} C_VEL
LIN {X 0,Y 544.641,Z 426.343,A -85,B 0,C 180,E1 -3466.269,E2 -3466.269} C_VEL
LIN {X 0,Y 544.616,Z 429.644,A -85,B 0,C 180,E1 -3467.352,E2 -3467.352} C_VEL
LIN {X 0,Y 544.593,Z 431.789,A -85,B 0,C 180,E1 -3468.458,E2 -3468.458} C_VEL
LIN {X 0,Y 544.545,Z 432.925,A -85,B 0,C 180,E1 -3469.81,E2 -3469.81} C_VEL
LIN {X 0,Y 544.548,Z 432.712,A -85,B 0,C 180,E1 -3470.772,E2 -3470.772} C_VEL
LIN {X 0,Y 544.536,Z 431.378,A -85,B 0,C 180,E1 -3471.931,E2 -3471.931} C_VEL
LIN {X 0,Y 544.614,Z 428.528,A -85,B 0,C 180,E1 -3473.136,E2 -3473.136} C_VEL
LIN {X 0,Y 544.658,Z 425.581,A -85,B 0,C 180,E1 -3474.009,E2 -3474.009} C_VEL
LIN {X 0,Y 544.695,Z 421.374,A -85,B 0,C 180,E1 -3474.958,E2 -3474.958} C_VEL
LIN {X 0,Y 544.749,Z 416.571,A -85,B 0,C 180,E1 -3475.817,E2 -3475.817} C_VEL
LIN {X 0,Y 544.833,Z 410.705,A -85,B 0,C 180,E1 -3476.666,E2 -3476.666} C_VEL
LIN {X 0,Y 544.933,Z 404.345,A -85,B 0,C 180,E1 -3477.421,E2 -3477.421} C_VEL
LIN {X 0,Y 545.029,Z 397.629,A -85,B 0,C 180,E1 -3478.083,E2 -3478.083} C_VEL
LIN {X 0,Y 545.109,Z 389.439,A -85,B 0,C 180,E1 -3478.748,E2 -3478.748} C_VEL
LIN {X 0,Y 545.293,Z 379.951,A -85,B 0,C 180,E1 -3479.363,E2 -3479.363} C_VEL
LIN {X 0,Y 545.435,Z 369.028,A -85,B 0,C 180,E1 -3479.886,E2 -3479.886} C_VEL
LIN {X 0,Y 545.422,Z 360.976,A -85,B 0,C 180,E1 -3480.178,E2 -3480.178} C_VEL
LIN {X 0,Y 544.61,Z 354.709,A -85,B 0,C 180,E1 -3480.382,E2 -3480.382} C_VEL
LIN {X 0,Y 544.609,Z 350.611,A -85,B 0,C 180,E1 -3483.149,E2 -3483.149} C_VEL
LIN {X 0,Y 544.626,Z 347.052,A -85,B 0,C 180,E1 -3485.61,E2 -3485.61} C_VEL
LIN {X 0,Y 544.64,Z 343.257,A -85,B 0,C 180,E1 -3488.289,E2 -3488.289} C_VEL
LIN {X 0,Y 544.686,Z 339.221,A -85,B 0,C 180,E1 -3491.181,E2 -3491.181} C_VEL
LIN {X 0,Y 544.723,Z 335.918,A -85,B 0,C 180,E1 -3493.509,E2 -3493.509} C_VEL
LIN {X 0,Y 544.749,Z 332.659,A -85,B 0,C 180,E1 -3495.81,E2 -3495.81} C_VEL
LIN {X 0,Y 544.896,Z 328.467,A -85,B 0,C 180,E1 -3498.844,E2 -3498.844} C_VEL
LIN {X 0,Y 544.889,Z 325.428,A -85,B 0,C 180,E1 -3501.095,E2 -3501.095} C_VEL
LIN {X 0,Y 545.091,Z 325.401,A -85,B 0,C 180,E1 -3503.336,E2 -3503.336} C_VEL
LIN {X 0,Y 545.197,Z 325.388,A -85,B 0,C 180,E1 -3504.822,E2 -3504.822} C_VEL
LIN {X 0,Y 545.183,Z 325.388,A -85,B 0,C 180,E1 -3507.783,E2 -3507.783} C_VEL
LIN {X 0,Y 545.206,Z 325.388,A -85,B 0,C 180,E1 -3510.738,E2 -3510.738} C_VEL
LIN {X 0,Y 545.166,Z 325.391,A -85,B 0,C 180,E1 -3512.955,E2 -3512.955} C_VEL
LIN {X 0,Y 545.163,Z 325.392,A -85,B 0,C 180,E1 -3515.919,E2 -3515.919} C_VEL
LIN {X 0,Y 545.118,Z 325.396,A -85,B 0,C 180,E1 -3518.899,E2 -3518.899} C_VEL
LIN {X 0,Y 545.124,Z 325.397,A -85,B 0,C 180,E1 -3521.903,E2 -3521.903} C_VEL
LIN {X 0,Y 545.073,Z 325.401,A -85,B 0,C 180,E1 -3524.943,E2 -3524.943} C_VEL
LIN {X 0,Y 545.071,Z 325.403,A -85,B 0,C 180,E1 -3528.025,E2 -3528.025} C_VEL
LIN {X 0,Y 545.088,Z 325.402,A -85,B 0,C 180,E1 -3530.371,E2 -3530.371} C_VEL
LIN {X 0,Y 545.078,Z 325.402,A -85,B 0,C 180,E1 -3533.558,E2 -3533.558} C_VEL
LIN {X 0,Y 545.075,Z 325.402,A -85,B 0,C 180,E1 -3535.999,E2 -3535.999} C_VEL
LIN {X 0,Y 545.08,Z 325.403,A -85,B 0,C 180,E1 -3538.749,E2 -3538.749} C_VEL
LIN {X 0,Y 545.064,Z 325.403,A -85,B 0,C 180,E1 -3541.682,E2 -3541.682} C_VEL
LIN {X 0,Y 545.072,Z 325.402,A -85,B 0,C 180,E1 -3544.562,E2 -3544.562} C_VEL
LIN {X 0,Y 545.055,Z 325.407,A -85,B 0,C 180,E1 -3547.301,E2 -3547.301} C_VEL
LIN {X 0,Y 545.08,Z 325.4,A -85,B 0,C 180,E1 -3550.14,E2 -3550.14} C_VEL
LIN {X 0,Y 545.053,Z 325.404,A -85,B 0,C 180,E1 -3552.697,E2 -3552.697} C_VEL
LIN {X 0,Y 545.048,Z 325.405,A -85,B 0,C 180,E1 -3555.167,E2 -3555.167} C_VEL
LIN {X 0,Y 545.067,Z 325.403,A -85,B 0,C 180,E1 -3557.898,E2 -3557.898} C_VEL
LIN {X 0,Y 545.093,Z 325.402,A -85,B 0,C 180,E1 -3560.675,E2 -3560.675} C_VEL
LIN {X 0,Y 545.046,Z 325.404,A -85,B 0,C 180,E1 -3563.621,E2 -3563.621} C_VEL
LIN {X 0,Y 545.064,Z 325.403,A -85,B 0,C 180,E1 -3566.329,E2 -3566.329} C_VEL
LIN {X 0,Y 545.056,Z 325.406,A -85,B 0,C 180,E1 -3568.953,E2 -3568.953} C_VEL
LIN {X 0,Y 545.092,Z 325.402,A -85,B 0,C 180,E1 -3571.508,E2 -3571.508} C_VEL
LIN {X 0,Y 545.081,Z 325.401,A -85,B 0,C 180,E1 -3574.491,E2 -3574.491} C_VEL
LIN {X 0,Y 545.055,Z 325.405,A -85,B 0,C 180,E1 -3577.244,E2 -3577.244} C_VEL
LIN {X 0,Y 545.108,Z 325.398,A -85,B 0,C 180,E1 -3580.415,E2 -3580.415} C_VEL
LIN {X 0,Y 545.066,Z 325.404,A -85,B 0,C 180,E1 -3583.522,E2 -3583.522} C_VEL
LIN {X 0,Y 545.083,Z 325.401,A -85,B 0,C 180,E1 -3585.821,E2 -3585.821} C_VEL
LIN {X 0,Y 545.105,Z 325.398,A -85,B 0,C 180,E1 -3588.85,E2 -3588.85} C_VEL
LIN {X 0,Y 545.123,Z 325.396,A -85,B 0,C 180,E1 -3591.848,E2 -3591.848} C_VEL
LIN {X 0,Y 545.198,Z 325.387,A -85,B 0,C 180,E1 -3594.824,E2 -3594.824} C_VEL
LIN {X 0,Y 545.19,Z 325.387,A -85,B 0,C 180,E1 -3597.784,E2 -3597.784} C_VEL
LIN {X 0,Y 545.208,Z 325.387,A -85,B 0,C 180,E1 -3600.739,E2 -3600.739} C_VEL
LIN {X 0,Y 545.165,Z 325.392,A -85,B 0,C 180,E1 -3602.957,E2 -3602.957} C_VEL
LIN {X 0,Y 545.161,Z 325.391,A -85,B 0,C 180,E1 -3605.92,E2 -3605.92} C_VEL
LIN {X 0,Y 545.11,Z 325.398,A -85,B 0,C 180,E1 -3608.901,E2 -3608.901} C_VEL
LIN {X 0,Y 545.127,Z 325.396,A -85,B 0,C 180,E1 -3611.905,E2 -3611.905} C_VEL
LIN {X 0,Y 545.076,Z 325.401,A -85,B 0,C 180,E1 -3614.944,E2 -3614.944} C_VEL
LIN {X 0,Y 545.074,Z 325.402,A -85,B 0,C 180,E1 -3618.026,E2 -3618.026} C_VEL
LIN {X 0,Y 545.087,Z 325.401,A -85,B 0,C 180,E1 -3620.373,E2 -3620.373} C_VEL
LIN {X 0,Y 545.083,Z 325.403,A -85,B 0,C 180,E1 -3623.56,E2 -3623.56} C_VEL
LIN {X 0,Y 545.081,Z 325.403,A -85,B 0,C 180,E1 -3626.001,E2 -3626.001} C_VEL
LIN {X 0,Y 545.086,Z 325.403,A -85,B 0,C 180,E1 -3628.75,E2 -3628.75} C_VEL
LIN {X 0,Y 545.061,Z 325.407,A -85,B 0,C 180,E1 -3631.049,E2 -3631.049} C_VEL
LIN {X 0,Y 545.071,Z 325.403,A -85,B 0,C 180,E1 -3633.672,E2 -3633.672} C_VEL
LIN {X 0,Y 545.049,Z 325.405,A -85,B 0,C 180,E1 -3636.38,E2 -3636.38} C_VEL
LIN {X 0,Y 545.098,Z 325.401,A -85,B 0,C 180,E1 -3639.325,E2 -3639.325} C_VEL
LIN {X 0,Y 545.077,Z 325.404,A -85,B 0,C 180,E1 -3642.103,E2 -3642.103} C_VEL
LIN {X 0,Y 545.058,Z 325.404,A -85,B 0,C 180,E1 -3645.168,E2 -3645.168} C_VEL
LIN {X 0,Y 545.078,Z 325.403,A -85,B 0,C 180,E1 -3647.899,E2 -3647.899} C_VEL
LIN {X 0,Y 545.079,Z 325.401,A -85,B 0,C 180,E1 -3650.82,E2 -3650.82} C_VEL
LIN {X 0,Y 545.052,Z 325.404,A -85,B 0,C 180,E1 -3653.622,E2 -3653.622} C_VEL
LIN {X 0,Y 545.171,Z 325.558,A -85,B 0,C 180,E1 -3655.819,E2 -3655.819} C_VEL
LIN {X 0,Y 545.67,Z 329.506,A -85,B 0,C 180,E1 -3657.254,E2 -3657.254} C_VEL
LIN {X 0,Y 545.568,Z 336.478,A -85,B 0,C 180,E1 -3659.666,E2 -3659.666} C_VEL
LIN {X 0,Y 545.339,Z 345.802,A -85,B 0,C 180,E1 -3662.777,E2 -3662.777} C_VEL
LIN {X 0,Y 545.201,Z 353.59,A -85,B 0,C 180,E1 -3665.233,E2 -3665.233} C_VEL
LIN {X 0,Y 545.114,Z 361.251,A -85,B 0,C 180,E1 -3667.647,E2 -3667.647} C_VEL
LIN {X 0,Y 544.987,Z 370.128,A -85,B 0,C 180,E1 -3670.411,E2 -3670.411} C_VEL
LIN {X 0,Y 544.901,Z 380.619,A -85,B 0,C 180,E1 -3673.517,E2 -3673.517} C_VEL
LIN {X 0,Y 544.831,Z 389.765,A -85,B 0,C 180,E1 -3676.195,E2 -3676.195} C_VEL
LIN {X 0,Y 544.754,Z 400.028,A -85,B 0,C 180,E1 -3679.219,E2 -3679.219} C_VEL
LIN {X 0,Y 544.743,Z 401.306,A -85,B 0,C 180,E1 -3679.595,E2 -3679.595} C_VEL
LIN {X 0,Y 545.548,Z 410.11,A -85,B 0,C 180,E1 -3679.845,E2 -3679.845} C_VEL
LIN {X 0,Y 545.445,Z 421.63,A -85,B 0,C 180,E1 -3680.265,E2 -3680.265} C_VEL
LIN {X 0,Y 545.257,Z 432.239,A -85,B 0,C 180,E1 -3680.823,E2 -3680.823} C_VEL
LIN {X 0,Y 545.153,Z 440.546,A -85,B 0,C 180,E1 -3681.382,E2 -3681.382} C_VEL
LIN {X 0,Y 545.035,Z 448.404,A -85,B 0,C 180,E1 -3682.033,E2 -3682.033} C_VEL
LIN {X 0,Y 544.92,Z 455.748,A -85,B 0,C 180,E1 -3682.777,E2 -3682.777} C_VEL
LIN {X 0,Y 544.854,Z 462.108,A -85,B 0,C 180,E1 -3683.563,E2 -3683.563} C_VEL
LIN {X 0,Y 544.711,Z 469.036,A -85,B 0,C 180,E1 -3684.634,E2 -3684.634} C_VEL
LIN {X 0,Y 544.706,Z 473.636,A -85,B 0,C 180,E1 -3685.561,E2 -3685.561} C_VEL
LIN {X 0,Y 544.675,Z 476.625,A -85,B 0,C 180,E1 -3686.302,E2 -3686.302} C_VEL
LIN {X 0,Y 544.658,Z 478.94,A -85,B 0,C 180,E1 -3687.042,E2 -3687.042} C_VEL
LIN {X 0,Y 544.572,Z 480.684,A -85,B 0,C 180,E1 -3687.782,E2 -3687.782} C_VEL
LIN {X 0,Y 544.545,Z 481.932,A -85,B 0,C 180,E1 -3688.522,E2 -3688.522} C_VEL
LIN {X 0,Y 544.538,Z 482.707,A -85,B 0,C 180,E1 -3689.261,E2 -3689.261} C_VEL
LIN {X 0,Y 544.538,Z 483,A -85,B 0,C 180,E1 -3690.001,E2 -3690.001} C_VEL
LIN {X 0,Y 544.538,Z 482.706,A -85,B 0,C 180,E1 -3690.74,E2 -3690.74} C_VEL
LIN {X 0,Y 544.545,Z 481.929,A -85,B 0,C 180,E1 -3691.48,E2 -3691.48} C_VEL
LIN {X 0,Y 544.572,Z 480.678,A -85,B 0,C 180,E1 -3692.22,E2 -3692.22} C_VEL
LIN {X 0,Y 544.687,Z 477.784,A -85,B 0,C 180,E1 -3693.33,E2 -3693.33} C_VEL
LIN {X 0,Y 544.696,Z 475.145,A -85,B 0,C 180,E1 -3694.07,E2 -3694.07} C_VEL
LIN {X 0,Y 544.671,Z 469.981,A -85,B 0,C 180,E1 -3695.183,E2 -3695.183} C_VEL
LIN {X 0,Y 544.881,Z 463.956,A -85,B 0,C 180,E1 -3696.183,E2 -3696.183} C_VEL
LIN {X 0,Y 544.923,Z 455.734,A -85,B 0,C 180,E1 -3697.225,E2 -3697.225} C_VEL
LIN {X 0,Y 545.038,Z 448.389,A -85,B 0,C 180,E1 -3697.969,E2 -3697.969} C_VEL
LIN {X 0,Y 545.155,Z 440.523,A -85,B 0,C 180,E1 -3698.62,E2 -3698.62} C_VEL
LIN {X 0,Y 545.261,Z 432.209,A -85,B 0,C 180,E1 -3699.179,E2 -3699.179} C_VEL
LIN {X 0,Y 545.451,Z 421.591,A -85,B 0,C 180,E1 -3699.737,E2 -3699.737} C_VEL
LIN {X 0,Y 545.578,Z 410.045,A -85,B 0,C 180,E1 -3700.156,E2 -3700.156} C_VEL
LIN {X 0,Y 544.742,Z 401.299,A -85,B 0,C 180,E1 -3700.407,E2 -3700.407} C_VEL
LIN {X 0,Y 544.809,Z 392.357,A -85,B 0,C 180,E1 -3703.048,E2 -3703.048} C_VEL
LIN {X 0,Y 544.892,Z 383.194,A -85,B 0,C 180,E1 -3705.716,E2 -3705.716} C_VEL
LIN {X 0,Y 544.952,Z 373.973,A -85,B 0,C 180,E1 -3708.42,E2 -3708.42} C_VEL
LIN {X 0,Y 545.029,Z 364.908,A -85,B 0,C 180,E1 -3711.166,E2 -3711.166} C_VEL
LIN {X 0,Y 545.14,Z 356.591,A -85,B 0,C 180,E1 -3713.746,E2 -3713.746} C_VEL
LIN {X 0,Y 545.271,Z 348.158,A -85,B 0,C 180,E1 -3716.403,E2 -3716.403} C_VEL
LIN {X 0,Y 545.48,Z 339.337,A -85,B 0,C 180,E1 -3719.315,E2 -3719.315} C_VEL
LIN {X 0,Y 545.678,Z 331.843,A -85,B 0,C 180,E1 -3721.875,E2 -3721.875} C_VEL
LIN {X 0,Y 545.594,Z 328.304,A -85,B 0,C 180,E1 -3723.145,E2 -3723.145} C_VEL
LIN {X 0,Y 545.102,Z 325.401,A -85,B 0,C 180,E1 -3724.253,E2 -3724.253} C_VEL
LIN {X 0,Y 545.041,Z 325.407,A -85,B 0,C 180,E1 -3727.304,E2 -3727.304} C_VEL
LIN {X 0,Y 545.069,Z 325.405,A -85,B 0,C 180,E1 -3730.143,E2 -3730.143} C_VEL
LIN {X 0,Y 545.084,Z 325.404,A -85,B 0,C 180,E1 -3733.107,E2 -3733.107} C_VEL
LIN {X 0,Y 545.055,Z 325.407,A -85,B 0,C 180,E1 -3736.227,E2 -3736.227} C_VEL
LIN {X 0,Y 545.087,Z 325.403,A -85,B 0,C 180,E1 -3738.886,E2 -3738.886} C_VEL
LIN {X 0,Y 545.053,Z 325.405,A -85,B 0,C 180,E1 -3741.865,E2 -3741.865} C_VEL
LIN {X 0,Y 545.042,Z 325.408,A -85,B 0,C 180,E1 -3744.532,E2 -3744.532} C_VEL
LIN {X 0,Y 545.07,Z 325.404,A -85,B 0,C 180,E1 -3747.211,E2 -3747.211} C_VEL
LIN {X 0,Y 545.067,Z 325.403,A -85,B 0,C 180,E1 -3749.81,E2 -3749.81} C_VEL
LIN {X 0,Y 545.09,Z 325.402,A -85,B 0,C 180,E1 -3752.829,E2 -3752.829} C_VEL
LIN {X 0,Y 545.055,Z 325.405,A -85,B 0,C 180,E1 -3755.631,E2 -3755.631} C_VEL
LIN {X 0,Y 545.071,Z 325.405,A -85,B 0,C 180,E1 -3758.836,E2 -3758.836} C_VEL
LIN {X 0,Y 545.079,Z 325.404,A -85,B 0,C 180,E1 -3761.195,E2 -3761.195} C_VEL
LIN {X 0,Y 545.07,Z 325.405,A -85,B 0,C 180,E1 -3763.521,E2 -3763.521} C_VEL
LIN {X 0,Y 545.097,Z 325.401,A -85,B 0,C 180,E1 -3765.819,E2 -3765.819} C_VEL
LIN {X 0,Y 545.123,Z 325.396,A -85,B 0,C 180,E1 -3768.849,E2 -3768.849} C_VEL
LIN {X 0,Y 545.103,Z 325.401,A -85,B 0,C 180,E1 -3771.846,E2 -3771.846} C_VEL
LIN {X 0,Y 545.207,Z 325.385,A -85,B 0,C 180,E1 -3774.822,E2 -3774.822} C_VEL
LIN {X 0,Y 545.196,Z 325.389,A -85,B 0,C 180,E1 -3777.783,E2 -3777.783} C_VEL
LIN {X 0,Y 545.218,Z 325.384,A -85,B 0,C 180,E1 -3780.738,E2 -3780.738} C_VEL
LIN {X 0,Y 545.173,Z 325.389,A -85,B 0,C 180,E1 -3782.955,E2 -3782.955} C_VEL
LIN {X 0,Y 545.173,Z 325.392,A -85,B 0,C 180,E1 -3785.919,E2 -3785.919} C_VEL
LIN {X 0,Y 545.101,Z 325.398,A -85,B 0,C 180,E1 -3788.899,E2 -3788.899} C_VEL
LIN {X 0,Y 545.138,Z 325.397,A -85,B 0,C 180,E1 -3791.903,E2 -3791.903} C_VEL
LIN {X 0,Y 545.089,Z 325.401,A -85,B 0,C 180,E1 -3794.943,E2 -3794.943} C_VEL
LIN {X 0,Y 545.067,Z 325.404,A -85,B 0,C 180,E1 -3797.417,E2 -3797.417} C_VEL
LIN {X 0,Y 544.864,Z 325.431,A -85,B 0,C 180,E1 -3798.811,E2 -3798.811} C_VEL
LIN {X 0,Y 544.834,Z 329.764,A -85,B 0,C 180,E1 -3801.966,E2 -3801.966} C_VEL
LIN {X 0,Y 544.786,Z 333.098,A -85,B 0,C 180,E1 -3804.381,E2 -3804.381} C_VEL
LIN {X 0,Y 544.737,Z 336.826,A -85,B 0,C 180,E1 -3807.099,E2 -3807.099} C_VEL
LIN {X 0,Y 544.671,Z 341.156,A -85,B 0,C 180,E1 -3810.172,E2 -3810.172} C_VEL
LIN {X 0,Y 544.634,Z 345.114,A -85,B 0,C 180,E1 -3812.989,E2 -3812.989} C_VEL
LIN {X 0,Y 544.582,Z 348.774,A -85,B 0,C 180,E1 -3815.606,E2 -3815.606} C_VEL
LIN {X 0,Y 544.561,Z 350.424,A -85,B 0,C 180,E1 -3816.766,E2 -3816.766} C_VEL
LIN {X 0,Y 543.883,Z 351.057,A -85,B 0,C 180,E1 -3817.172,E2 -3817.172} C_VEL
LIN {X 0,Y 541.003,Z 352.174,A -85,B 0,C 180,E1 -3817.806,E2 -3817.806} C_VEL
LIN {X 0,Y 538.124,Z 353.295,A -85,B 0,C 180,E1 -3818.445,E2 -3818.445} C_VEL
LIN {X 0,Y 537.463,Z 353.934,A -85,B 0,C 180,E1 -3818.859,E2 -3818.859} C_VEL
LIN {X 0,Y 537.493,Z 354.955,A -85,B 0,C 180,E1 -3819.57,E2 -3819.57} C_VEL
LIN {X 0,Y 538.573,Z 363.897,A -85,B 0,C 180,E1 -3819.868,E2 -3819.868} C_VEL
LIN {X 0,Y 538.396,Z 374.431,A -85,B 0,C 180,E1 -3820.312,E2 -3820.312} C_VEL
LIN {X 0,Y 538.262,Z 382.796,A -85,B 0,C 180,E1 -3820.773,E2 -3820.773} C_VEL
LIN {X 0,Y 538.067,Z 391.72,A -85,B 0,C 180,E1 -3821.393,E2 -3821.393} C_VEL
LIN {X 0,Y 537.967,Z 399.465,A -85,B 0,C 180,E1 -3822.062,E2 -3822.062} C_VEL
LIN {X 0,Y 537.836,Z 407.921,A -85,B 0,C 180,E1 -3822.965,E2 -3822.965} C_VEL
LIN {X 0,Y 537.712,Z 414.384,A -85,B 0,C 180,E1 -3823.844,E2 -3823.844} C_VEL
LIN {X 0,Y 537.64,Z 420.517,A -85,B 0,C 180,E1 -3824.899,E2 -3824.899} C_VEL
LIN {X 0,Y 537.587,Z 423.694,A -85,B 0,C 180,E1 -3825.561,E2 -3825.561} C_VEL
LIN {X 0,Y 537.559,Z 427.661,A -85,B 0,C 180,E1 -3826.631,E2 -3826.631} C_VEL
LIN {X 0,Y 537.541,Z 429.282,A -85,B 0,C 180,E1 -3827.166,E2 -3827.166} C_VEL
LIN {X 0,Y 537.496,Z 431.454,A -85,B 0,C 180,E1 -3828.183,E2 -3828.183} C_VEL
LIN {X 0,Y 537.457,Z 432.718,A -85,B 0,C 180,E1 -3829.324,E2 -3829.324} C_VEL
LIN {X 0,Y 537.427,Z 432.835,A -85,B 0,C 180,E1 -3830.491,E2 -3830.491} C_VEL
LIN {X 0,Y 537.427,Z 432.473,A -85,B 0,C 180,E1 -3831.118,E2 -3831.118} C_VEL
LIN {X 0,Y 537.439,Z 431.149,A -85,B 0,C 180,E1 -3832.076,E2 -3832.076} C_VEL
LIN {X 0,Y 537.505,Z 428.994,A -85,B 0,C 180,E1 -3833.025,E2 -3833.025} C_VEL
LIN {X 0,Y 537.571,Z 425.228,A -85,B 0,C 180,E1 -3834.149,E2 -3834.149} C_VEL
LIN {X 0,Y 537.627,Z 420.536,A -85,B 0,C 180,E1 -3835.188,E2 -3835.188} C_VEL
LIN {X 0,Y 537.673,Z 415.745,A -85,B 0,C 180,E1 -3836.027,E2 -3836.027} C_VEL
LIN {X 0,Y 537.811,Z 409.2,A -85,B 0,C 180,E1 -3836.959,E2 -3836.959} C_VEL
LIN {X 0,Y 537.94,Z 400.907,A -85,B 0,C 180,E1 -3837.893,E2 -3837.893} C_VEL
LIN {X 0,Y 538.066,Z 392.818,A -85,B 0,C 180,E1 -3838.611,E2 -3838.611} C_VEL
LIN {X 0,Y 538.152,Z 385.25,A -85,B 0,C 180,E1 -3839.163,E2 -3839.163} C_VEL
LIN {X 0,Y 538.296,Z 376.757,A -85,B 0,C 180,E1 -3839.661,E2 -3839.661} C_VEL
LIN {X 0,Y 538.468,Z 368.295,A -85,B 0,C 180,E1 -3840.05,E2 -3840.05} C_VEL
LIN {X 0,Y 538.34,Z 361.204,A -85,B 0,C 180,E1 -3840.311,E2 -3840.311} C_VEL
LIN {X 0,Y 537.528,Z 354.888,A -85,B 0,C 180,E1 -3840.531,E2 -3840.531} C_VEL
LIN {X 0,Y 537.52,Z 350.401,A -85,B 0,C 180,E1 -3843.605,E2 -3843.605} C_VEL
LIN {X 0,Y 537.562,Z 346.67,A -85,B 0,C 180,E1 -3846.226,E2 -3846.226} C_VEL
LIN {X 0,Y 537.56,Z 342.39,A -85,B 0,C 180,E1 -3849.329,E2 -3849.329} C_VEL
LIN {X 0,Y 537.614,Z 339.013,A -85,B 0,C 180,E1 -3851.714,E2 -3851.714} C_VEL
LIN {X 0,Y 537.633,Z 335.754,A -85,B 0,C 180,E1 -3854.066,E2 -3854.066} C_VEL
LIN {X 0,Y 537.658,Z 332.518,A -85,B 0,C 180,E1 -3856.391,E2 -3856.391} C_VEL
LIN {X 0,Y 537.847,Z 329.37,A -85,B 0,C 180,E1 -3858.696,E2 -3858.696} C_VEL
LIN {X 0,Y 537.81,Z 326.31,A -85,B 0,C 180,E1 -3860.977,E2 -3860.977} C_VEL
LIN {X 0,Y 538.061,Z 326.276,A -85,B 0,C 180,E1 -3863.248,E2 -3863.248} C_VEL
LIN {X 0,Y 538.154,Z 326.266,A -85,B 0,C 180,E1 -3864.754,E2 -3864.754} C_VEL
LIN {X 0,Y 538.155,Z 326.264,A -85,B 0,C 180,E1 -3867.754,E2 -3867.754} C_VEL
LIN {X 0,Y 538.175,Z 326.264,A -85,B 0,C 180,E1 -3870.747,E2 -3870.747} C_VEL
LIN {X 0,Y 538.132,Z 326.267,A -85,B 0,C 180,E1 -3872.993,E2 -3872.993} C_VEL
LIN {X 0,Y 538.115,Z 326.269,A -85,B 0,C 180,E1 -3875.996,E2 -3875.996} C_VEL
LIN {X 0,Y 538.068,Z 326.275,A -85,B 0,C 180,E1 -3879.017,E2 -3879.017} C_VEL
LIN {X 0,Y 538.072,Z 326.275,A -85,B 0,C 180,E1 -3882.062,E2 -3882.062} C_VEL
LIN {X 0,Y 538.033,Z 326.279,A -85,B 0,C 180,E1 -3885.143,E2 -3885.143} C_VEL
LIN {X 0,Y 538.023,Z 326.28,A -85,B 0,C 180,E1 -3888.269,E2 -3888.269} C_VEL
LIN {X 0,Y 538.031,Z 326.279,A -85,B 0,C 180,E1 -3890.65,E2 -3890.65} C_VEL
LIN {X 0,Y 538.01,Z 326.284,A -85,B 0,C 180,E1 -3893.887,E2 -3893.887} C_VEL
LIN {X 0,Y 538.037,Z 326.28,A -85,B 0,C 180,E1 -3896.366,E2 -3896.366} C_VEL
LIN {X 0,Y 538.042,Z 326.28,A -85,B 0,C 180,E1 -3898.938,E2 -3898.938} C_VEL
LIN {X 0,Y 538.014,Z 326.281,A -85,B 0,C 180,E1 -3901.89,E2 -3901.89} C_VEL
LIN {X 0,Y 538.022,Z 326.281,A -85,B 0,C 180,E1 -3904.621,E2 -3904.621} C_VEL
LIN {X 0,Y 538.011,Z 326.284,A -85,B 0,C 180,E1 -3907.173,E2 -3907.173} C_VEL
LIN {X 0,Y 538.041,Z 326.279,A -85,B 0,C 180,E1 -3909.794,E2 -3909.794} C_VEL
LIN {X 0,Y 538.011,Z 326.282,A -85,B 0,C 180,E1 -3912.785,E2 -3912.785} C_VEL
LIN {X 0,Y 538.013,Z 326.283,A -85,B 0,C 180,E1 -3915.925,E2 -3915.925} C_VEL
LIN {X 0,Y 538.063,Z 326.277,A -85,B 0,C 180,E1 -3919.249,E2 -3919.249} C_VEL
LIN {X 0,Y 537.989,Z 326.285,A -85,B 0,C 180,E1 -3922.123,E2 -3922.123} C_VEL
LIN {X 0,Y 538.008,Z 326.282,A -85,B 0,C 180,E1 -3924.918,E2 -3924.918} C_VEL
LIN {X 0,Y 538.017,Z 326.282,A -85,B 0,C 180,E1 -3927.618,E2 -3927.618} C_VEL
LIN {X 0,Y 538.029,Z 326.281,A -85,B 0,C 180,E1 -3930.241,E2 -3930.241} C_VEL
LIN {X 0,Y 538.053,Z 326.279,A -85,B 0,C 180,E1 -3932.797,E2 -3932.797} C_VEL
LIN {X 0,Y 538.041,Z 326.279,A -85,B 0,C 180,E1 -3935.293,E2 -3935.293} C_VEL
LIN {X 0,Y 538.018,Z 326.281,A -85,B 0,C 180,E1 -3938.038,E2 -3938.038} C_VEL
LIN {X 0,Y 538.029,Z 326.28,A -85,B 0,C 180,E1 -3940.941,E2 -3940.941} C_VEL
LIN {X 0,Y 538.016,Z 326.281,A -85,B 0,C 180,E1 -3943.3,E2 -3943.3} C_VEL
LIN {X 0,Y 538.051,Z 326.276,A -85,B 0,C 180,E1 -3945.631,E2 -3945.631} C_VEL
LIN {X 0,Y 538.064,Z 326.276,A -85,B 0,C 180,E1 -3948.702,E2 -3948.702} C_VEL
LIN {X 0,Y 538.08,Z 326.273,A -85,B 0,C 180,E1 -3951.74,E2 -3951.74} C_VEL
LIN {X 0,Y 538.155,Z 326.265,A -85,B 0,C 180,E1 -3954.756,E2 -3954.756} C_VEL
LIN {X 0,Y 538.161,Z 326.263,A -85,B 0,C 180,E1 -3957.755,E2 -3957.755} C_VEL
LIN {X 0,Y 538.178,Z 326.262,A -85,B 0,C 180,E1 -3960.749,E2 -3960.749} C_VEL
LIN {X 0,Y 538.132,Z 326.268,A -85,B 0,C 180,E1 -3962.995,E2 -3962.995} C_VEL
LIN {X 0,Y 538.114,Z 326.269,A -85,B 0,C 180,E1 -3965.998,E2 -3965.998} C_VEL
LIN {X 0,Y 538.061,Z 326.276,A -85,B 0,C 180,E1 -3969.018,E2 -3969.018} C_VEL
LIN {X 0,Y 538.075,Z 326.274,A -85,B 0,C 180,E1 -3972.063,E2 -3972.063} C_VEL
LIN {X 0,Y 538.036,Z 326.28,A -85,B 0,C 180,E1 -3975.145,E2 -3975.145} C_VEL
LIN {X 0,Y 538.026,Z 326.279,A -85,B 0,C 180,E1 -3978.271,E2 -3978.271} C_VEL
LIN {X 0,Y 538.031,Z 326.278,A -85,B 0,C 180,E1 -3980.652,E2 -3980.652} C_VEL
LIN {X 0,Y 538.015,Z 326.282,A -85,B 0,C 180,E1 -3983.888,E2 -3983.888} C_VEL
LIN {X 0,Y 538.042,Z 326.279,A -85,B 0,C 180,E1 -3986.367,E2 -3986.367} C_VEL
LIN {X 0,Y 538.048,Z 326.278,A -85,B 0,C 180,E1 -3988.94,E2 -3988.94} C_VEL
LIN {X 0,Y 538.006,Z 326.283,A -85,B 0,C 180,E1 -3991.889,E2 -3991.889} C_VEL
LIN {X 0,Y 538.028,Z 326.281,A -85,B 0,C 180,E1 -3994.622,E2 -3994.622} C_VEL
LIN {X 0,Y 538.001,Z 326.285,A -85,B 0,C 180,E1 -3997.172,E2 -3997.172} C_VEL
LIN {X 0,Y 538.021,Z 326.281,A -85,B 0,C 180,E1 -3999.798,E2 -3999.798} C_VEL
LIN {X 0,Y 538.018,Z 326.281,A -85,B 0,C 180,E1 -4002.787,E2 -4002.787} C_VEL
LIN {X 0,Y 538.023,Z 326.28,A -85,B 0,C 180,E1 -4005.927,E2 -4005.927} C_VEL
LIN {X 0,Y 538.047,Z 326.28,A -85,B 0,C 180,E1 -4009.226,E2 -4009.226} C_VEL
LIN {X 0,Y 537.99,Z 326.284,A -85,B 0,C 180,E1 -4012.124,E2 -4012.124} C_VEL
LIN {X 0,Y 538.108,Z 326.272,A -85,B 0,C 180,E1 -4015.495,E2 -4015.495} C_VEL
LIN {X 0,Y 538.39,Z 328.137,A -85,B 0,C 180,E1 -4016.28,E2 -4016.28} C_VEL
LIN {X 0,Y 538.71,Z 332.871,A -85,B 0,C 180,E1 -4017.994,E2 -4017.994} C_VEL
LIN {X 0,Y 538.444,Z 341.958,A -85,B 0,C 180,E1 -4021.124,E2 -4021.124} C_VEL
LIN {X 0,Y 538.285,Z 349.597,A -85,B 0,C 180,E1 -4023.647,E2 -4023.647} C_VEL
LIN {X 0,Y 538.15,Z 358.544,A -85,B 0,C 180,E1 -4026.528,E2 -4026.528} C_VEL
LIN {X 0,Y 537.986,Z 368.699,A -85,B 0,C 180,E1 -4029.747,E2 -4029.747} C_VEL
LIN {X 0,Y 537.866,Z 377.816,A -85,B 0,C 180,E1 -4032.526,E2 -4032.526} C_VEL
LIN {X 0,Y 537.776,Z 388.234,A -85,B 0,C 180,E1 -4035.624,E2 -4035.624} C_VEL
LIN {X 0,Y 537.692,Z 398.649,A -85,B 0,C 180,E1 -4038.694,E2 -4038.694} C_VEL
LIN {X 0,Y 537.656,Z 401.245,A -85,B 0,C 180,E1 -4039.456,E2 -4039.456} C_VEL
LIN {X 0,Y 538.566,Z 410.901,A -85,B 0,C 180,E1 -4039.736,E2 -4039.736} C_VEL
LIN {X 0,Y 538.451,Z 421.62,A -85,B 0,C 180,E1 -4040.137,E2 -4040.137} C_VEL
LIN {X 0,Y 538.26,Z 432.237,A -85,B 0,C 180,E1 -4040.703,E2 -4040.703} C_VEL
LIN {X 0,Y 538.135,Z 440.543,A -85,B 0,C 180,E1 -4041.269,E2 -4041.269} C_VEL
LIN {X 0,Y 537.985,Z 448.402,A -85,B 0,C 180,E1 -4041.928,E2 -4041.928} C_VEL
LIN {X 0,Y 537.852,Z 455.747,A -85,B 0,C 180,E1 -4042.682,E2 -4042.682} C_VEL
LIN {X 0,Y 537.789,Z 462.695,A -85,B 0,C 180,E1 -4043.556,E2 -4043.556} C_VEL
LIN {X 0,Y 537.651,Z 469.036,A -85,B 0,C 180,E1 -4044.563,E2 -4044.563} C_VEL
LIN {X 0,Y 537.607,Z 473.636,A -85,B 0,C 180,E1 -4045.502,E2 -4045.502} C_VEL
LIN {X 0,Y 537.598,Z 476.624,A -85,B 0,C 180,E1 -4046.253,E2 -4046.253} C_VEL
LIN {X 0,Y 537.562,Z 478.941,A -85,B 0,C 180,E1 -4047.003,E2 -4047.003} C_VEL
LIN {X 0,Y 537.491,Z 480.683,A -85,B 0,C 180,E1 -4047.753,E2 -4047.753} C_VEL
LIN {X 0,Y 537.45,Z 481.93,A -85,B 0,C 180,E1 -4048.502,E2 -4048.502} C_VEL
LIN {X 0,Y 537.438,Z 482.707,A -85,B 0,C 180,E1 -4049.252,E2 -4049.252} C_VEL
LIN {X 0,Y 537.439,Z 483,A -85,B 0,C 180,E1 -4050.001,E2 -4050.001} C_VEL
LIN {X 0,Y 537.438,Z 482.706,A -85,B 0,C 180,E1 -4050.75,E2 -4050.75} C_VEL
LIN {X 0,Y 537.45,Z 481.927,A -85,B 0,C 180,E1 -4051.5,E2 -4051.5} C_VEL
LIN {X 0,Y 537.491,Z 480.677,A -85,B 0,C 180,E1 -4052.249,E2 -4052.249} C_VEL
LIN {X 0,Y 537.587,Z 477.783,A -85,B 0,C 180,E1 -4053.374,E2 -4053.374} C_VEL
LIN {X 0,Y 537.62,Z 475.145,A -85,B 0,C 180,E1 -4054.124,E2 -4054.124} C_VEL
LIN {X 0,Y 537.604,Z 469.981,A -85,B 0,C 180,E1 -4055.251,E2 -4055.251} C_VEL
LIN {X 0,Y 537.803,Z 464.199,A -85,B 0,C 180,E1 -4056.226,E2 -4056.226} C_VEL
LIN {X 0,Y 537.855,Z 457.427,A -85,B 0,C 180,E1 -4057.132,E2 -4057.132} C_VEL
LIN {X 0,Y 537.992,Z 449.408,A -85,B 0,C 180,E1 -4057.979,E2 -4057.979} C_VEL
LIN {X 0,Y 538.129,Z 441.751,A -85,B 0,C 180,E1 -4058.639,E2 -4058.639} C_VEL
LIN {X 0,Y 538.22,Z 433.707,A -85,B 0,C 180,E1 -4059.205,E2 -4059.205} C_VEL
LIN {X 0,Y 538.373,Z 425.369,A -85,B 0,C 180,E1 -4059.677,E2 -4059.677} C_VEL
LIN {X 0,Y 538.47,Z 416.837,A -85,B 0,C 180,E1 -4060.054,E2 -4060.054} C_VEL
LIN {X 0,Y 538.504,Z 407.91,A -85,B 0,C 180,E1 -4060.351,E2 -4060.351} C_VEL
LIN {X 0,Y 537.65,Z 401.228,A -85,B 0,C 180,E1 -4060.546,E2 -4060.546} C_VEL
LIN {X 0,Y 537.711,Z 392.096,A -85,B 0,C 180,E1 -4063.223,E2 -4063.223} C_VEL
LIN {X 0,Y 537.821,Z 384.234,A -85,B 0,C 180,E1 -4065.539,E2 -4065.539} C_VEL
LIN {X 0,Y 537.896,Z 373.695,A -85,B 0,C 180,E1 -4068.67,E2 -4068.67} C_VEL
LIN {X 0,Y 537.995,Z 364.694,A -85,B 0,C 180,E1 -4071.456,E2 -4071.456} C_VEL
LIN {X 0,Y 538.155,Z 354.398,A -85,B 0,C 180,E1 -4074.703,E2 -4074.703} C_VEL
LIN {X 0,Y 538.294,Z 346.132,A -85,B 0,C 180,E1 -4077.4,E2 -4077.4} C_VEL
LIN {X 0,Y 538.533,Z 338.028,A -85,B 0,C 180,E1 -4080.136,E2 -4080.136} C_VEL
LIN {X 0,Y 538.661,Z 330.589,A -85,B 0,C 180,E1 -4082.784,E2 -4082.784} C_VEL
LIN {X 0,Y 538.051,Z 326.279,A -85,B 0,C 180,E1 -4084.506,E2 -4084.506} C_VEL
LIN {X 0,Y 538.009,Z 326.284,A -85,B 0,C 180,E1 -4087.17,E2 -4087.17} C_VEL
LIN {X 0,Y 538.026,Z 326.282,A -85,B 0,C 180,E1 -4089.798,E2 -4089.798} C_VEL
LIN {X 0,Y 538.025,Z 326.285,A -85,B 0,C 180,E1 -4092.786,E2 -4092.786} C_VEL
LIN {X 0,Y 538.01,Z 326.286,A -85,B 0,C 180,E1 -4095.138,E2 -4095.138} C_VEL
LIN {X 0,Y 538.036,Z 326.279,A -85,B 0,C 180,E1 -4098.227,E2 -4098.227} C_VEL
LIN {X 0,Y 538.016,Z 326.284,A -85,B 0,C 180,E1 -4101.169,E2 -4101.169} C_VEL
LIN {X 0,Y 538,Z 326.283,A -85,B 0,C 180,E1 -4104.089,E2 -4104.089} C_VEL
LIN {X 0,Y 538.037,Z 326.279,A -85,B 0,C 180,E1 -4106.727,E2 -4106.727} C_VEL
LIN {X 0,Y 538.02,Z 326.282,A -85,B 0,C 180,E1 -4109.559,E2 -4109.559} C_VEL
LIN {X 0,Y 538.054,Z 326.277,A -85,B 0,C 180,E1 -4112.65,E2 -4112.65} C_VEL
LIN {X 0,Y 538.054,Z 326.279,A -85,B 0,C 180,E1 -4115.292,E2 -4115.292} C_VEL
LIN {X 0,Y 538.028,Z 326.28,A -85,B 0,C 180,E1 -4118.546,E2 -4118.546} C_VEL
LIN {X 0,Y 538.037,Z 326.279,A -85,B 0,C 180,E1 -4120.94,E2 -4120.94} C_VEL
LIN {X 0,Y 538.018,Z 326.281,A -85,B 0,C 180,E1 -4123.298,E2 -4123.298} C_VEL
LIN {X 0,Y 538.067,Z 326.276,A -85,B 0,C 180,E1 -4125.63,E2 -4125.63} C_VEL
LIN {X 0,Y 538.083,Z 326.273,A -85,B 0,C 180,E1 -4128.701,E2 -4128.701} C_VEL
LIN {X 0,Y 538.067,Z 326.277,A -85,B 0,C 180,E1 -4131.739,E2 -4131.739} C_VEL
LIN {X 0,Y 538.164,Z 326.262,A -85,B 0,C 180,E1 -4134.754,E2 -4134.754} C_VEL
LIN {X 0,Y 538.168,Z 326.264,A -85,B 0,C 180,E1 -4137.754,E2 -4137.754} C_VEL
LIN {X 0,Y 538.188,Z 326.259,A -85,B 0,C 180,E1 -4140.747,E2 -4140.747} C_VEL
LIN {X 0,Y 538.14,Z 326.265,A -85,B 0,C 180,E1 -4142.994,E2 -4142.994} C_VEL
LIN {X 0,Y 538.126,Z 326.27,A -85,B 0,C 180,E1 -4145.996,E2 -4145.996} C_VEL
LIN {X 0,Y 538.055,Z 326.276,A -85,B 0,C 180,E1 -4149.017,E2 -4149.017} C_VEL
LIN {X 0,Y 538.087,Z 326.274,A -85,B 0,C 180,E1 -4152.062,E2 -4152.062} C_VEL
LIN {X 0,Y 538.048,Z 326.279,A -85,B 0,C 180,E1 -4155.143,E2 -4155.143} C_VEL
LIN {X 0,Y 538.014,Z 326.284,A -85,B 0,C 180,E1 -4157.523,E2 -4157.523} C_VEL
LIN {X 0,Y 537.794,Z 326.512,A -85,B 0,C 180,E1 -4159.068,E2 -4159.068} C_VEL
LIN {X 0,Y 537.773,Z 330.371,A -85,B 0,C 180,E1 -4161.892,E2 -4161.892} C_VEL
LIN {X 0,Y 537.741,Z 334.221,A -85,B 0,C 180,E1 -4164.721,E2 -4164.721} C_VEL
LIN {X 0,Y 537.657,Z 337.735,A -85,B 0,C 180,E1 -4167.268,E2 -4167.268} C_VEL
LIN {X 0,Y 537.596,Z 342.05,A -85,B 0,C 180,E1 -4170.364,E2 -4170.364} C_VEL
LIN {X 0,Y 537.546,Z 346.144,A -85,B 0,C 180,E1 -4173.305,E2 -4173.305} C_VEL
LIN {X 0,Y 537.49,Z 349.936,A -85,B 0,C 180,E1 -4176.042,E2 -4176.042} C_VEL
LIN {X 0,Y 537.463,Z 353.934,A -85,B 0,C 180,E1 -4178.859,E2 -4178.859} C_VEL
LIN {X 0,Y 537.301,Z 355.068,A -85,B 0,C 180,E1 -4179.153,E2 -4179.153} C_VEL
LIN {X 0,Y 536.696,Z 357.91,A -85,B 0,C 180,E1 -4179.459,E2 -4179.459} C_VEL
LIN {X 0,Y 535.535,Z 362.616,A -85,B 0,C 180,E1 -4179.728,E2 -4179.728} C_VEL
LIN {X 0,Y 532.356,Z 373.983,A -85,B 0,C 180,E1 -4180.163,E2 -4180.163} C_VEL
LIN {X 0,Y 531.41,Z 379.209,A -85,B 0,C 180,E1 -4180.411,E2 -4180.411} C_VEL
LIN {X 0,Y 531.345,Z 380.908,A -85,B 0,C 180,E1 -4180.51,E2 -4180.51} C_VEL
LIN {X 0,Y 531.129,Z 390.082,A -85,B 0,C 180,E1 -4181.125,E2 -4181.125} C_VEL
LIN {X 0,Y 530.98,Z 398.302,A -85,B 0,C 180,E1 -4181.816,E2 -4181.816} C_VEL
LIN {X 0,Y 530.859,Z 404.701,A -85,B 0,C 180,E1 -4182.467,E2 -4182.467} C_VEL
LIN {X 0,Y 530.759,Z 411.139,A -85,B 0,C 180,E1 -4183.257,E2 -4183.257} C_VEL
LIN {X 0,Y 530.61,Z 416.991,A -85,B 0,C 180,E1 -4184.134,E2 -4184.134} C_VEL
LIN {X 0,Y 530.568,Z 421.651,A -85,B 0,C 180,E1 -4184.996,E2 -4184.996} C_VEL
LIN {X 0,Y 530.483,Z 426.212,A -85,B 0,C 180,E1 -4186.064,E2 -4186.064} C_VEL
LIN {X 0,Y 530.463,Z 428.489,A -85,B 0,C 180,E1 -4186.774,E2 -4186.774} C_VEL
LIN {X 0,Y 530.413,Z 431.2,A -85,B 0,C 180,E1 -4187.9,E2 -4187.9} C_VEL
LIN {X 0,Y 530.376,Z 432.797,A -85,B 0,C 180,E1 -4189.05,E2 -4189.05} C_VEL
LIN {X 0,Y 530.35,Z 433.057,A -85,B 0,C 180,E1 -4190.499,E2 -4190.499} C_VEL
LIN {X 0,Y 530.332,Z 432.27,A -85,B 0,C 180,E1 -4191.475,E2 -4191.475} C_VEL
LIN {X 0,Y 530.376,Z 430.209,A -85,B 0,C 180,E1 -4192.659,E2 -4192.659} C_VEL
LIN {X 0,Y 530.485,Z 426.638,A -85,B 0,C 180,E1 -4193.913,E2 -4193.913} C_VEL
LIN {X 0,Y 530.547,Z 421.918,A -85,B 0,C 180,E1 -4195.039,E2 -4195.039} C_VEL
LIN {X 0,Y 530.605,Z 416.896,A -85,B 0,C 180,E1 -4195.97,E2 -4195.97} C_VEL
LIN {X 0,Y 530.733,Z 411.151,A -85,B 0,C 180,E1 -4196.83,E2 -4196.83} C_VEL
LIN {X 0,Y 530.876,Z 403.433,A -85,B 0,C 180,E1 -4197.763,E2 -4197.763} C_VEL
LIN {X 0,Y 531.053,Z 393.379,A -85,B 0,C 180,E1 -4198.705,E2 -4198.705} C_VEL
LIN {X 0,Y 531.165,Z 385.017,A -85,B 0,C 180,E1 -4199.318,E2 -4199.318} C_VEL
LIN {X 0,Y 531.346,Z 376.306,A -85,B 0,C 180,E1 -4199.826,E2 -4199.826} C_VEL
LIN {X 0,Y 531.484,Z 367.715,A -85,B 0,C 180,E1 -4200.217,E2 -4200.217} C_VEL
LIN {X 0,Y 531.39,Z 362.095,A -85,B 0,C 180,E1 -4200.429,E2 -4200.429} C_VEL
LIN {X 0,Y 530.479,Z 355.209,A -85,B 0,C 180,E1 -4200.671,E2 -4200.671} C_VEL
LIN {X 0,Y 530.431,Z 351.531,A -85,B 0,C 180,E1 -4203.224,E2 -4203.224} C_VEL
LIN {X 0,Y 530.515,Z 347.519,A -85,B 0,C 180,E1 -4206.072,E2 -4206.072} C_VEL
LIN {X 0,Y 530.496,Z 343.355,A -85,B 0,C 180,E1 -4209.04,E2 -4209.04} C_VEL
LIN {X 0,Y 530.525,Z 339.96,A -85,B 0,C 180,E1 -4211.461,E2 -4211.461} C_VEL
LIN {X 0,Y 530.566,Z 336.663,A -85,B 0,C 180,E1 -4213.848,E2 -4213.848} C_VEL
LIN {X 0,Y 530.603,Z 333.434,A -85,B 0,C 180,E1 -4216.206,E2 -4216.206} C_VEL
LIN {X 0,Y 530.774,Z 329.175,A -85,B 0,C 180,E1 -4219.316,E2 -4219.316} C_VEL
LIN {X 0,Y 530.741,Z 327.19,A -85,B 0,C 180,E1 -4220.856,E2 -4220.856} C_VEL
LIN {X 0,Y 531.045,Z 327.149,A -85,B 0,C 180,E1 -4223.158,E2 -4223.158} C_VEL
LIN {X 0,Y 530.994,Z 327.155,A -85,B 0,C 180,E1 -4225.444,E2 -4225.444} C_VEL
LIN {X 0,Y 531.128,Z 327.139,A -85,B 0,C 180,E1 -4227.724,E2 -4227.724} C_VEL
LIN {X 0,Y 531.145,Z 327.139,A -85,B 0,C 180,E1 -4230.757,E2 -4230.757} C_VEL
LIN {X 0,Y 531.099,Z 327.144,A -85,B 0,C 180,E1 -4233.033,E2 -4233.033} C_VEL
LIN {X 0,Y 531.075,Z 327.146,A -85,B 0,C 180,E1 -4236.076,E2 -4236.076} C_VEL
LIN {X 0,Y 531.027,Z 327.152,A -85,B 0,C 180,E1 -4239.137,E2 -4239.137} C_VEL
LIN {X 0,Y 531.029,Z 327.151,A -85,B 0,C 180,E1 -4242.224,E2 -4242.224} C_VEL
LIN {X 0,Y 530.984,Z 327.159,A -85,B 0,C 180,E1 -4245.349,E2 -4245.349} C_VEL
LIN {X 0,Y 531.003,Z 327.157,A -85,B 0,C 180,E1 -4247.722,E2 -4247.722} C_VEL
LIN {X 0,Y 530.99,Z 327.155,A -85,B 0,C 180,E1 -4250.937,E2 -4250.937} C_VEL
LIN {X 0,Y 530.966,Z 327.159,A -85,B 0,C 180,E1 -4254.224,E2 -4254.224} C_VEL
LIN {X 0,Y 530.998,Z 327.155,A -85,B 0,C 180,E1 -4256.743,E2 -4256.743} C_VEL
LIN {X 0,Y 530.986,Z 327.157,A -85,B 0,C 180,E1 -4259.321,E2 -4259.321} C_VEL
LIN {X 0,Y 530.966,Z 327.16,A -85,B 0,C 180,E1 -4262.103,E2 -4262.103} C_VEL
LIN {X 0,Y 530.978,Z 327.16,A -85,B 0,C 180,E1 -4264.854,E2 -4264.854} C_VEL
LIN {X 0,Y 530.959,Z 327.161,A -85,B 0,C 180,E1 -4267.507,E2 -4267.507} C_VEL
LIN {X 0,Y 530.995,Z 327.155,A -85,B 0,C 180,E1 -4270.43,E2 -4270.43} C_VEL
LIN {X 0,Y 530.953,Z 327.162,A -85,B 0,C 180,E1 -4273.494,E2 -4273.494} C_VEL
LIN {X 0,Y 530.951,Z 327.161,A -85,B 0,C 180,E1 -4276.506,E2 -4276.506} C_VEL
LIN {X 0,Y 530.993,Z 327.156,A -85,B 0,C 180,E1 -4279.57,E2 -4279.57} C_VEL
LIN {X 0,Y 530.963,Z 327.16,A -85,B 0,C 180,E1 -4282.576,E2 -4282.576} C_VEL
LIN {X 0,Y 530.99,Z 327.158,A -85,B 0,C 180,E1 -4285.312,E2 -4285.312} C_VEL
LIN {X 0,Y 530.968,Z 327.161,A -85,B 0,C 180,E1 -4288.033,E2 -4288.033} C_VEL
LIN {X 0,Y 530.993,Z 327.156,A -85,B 0,C 180,E1 -4290.871,E2 -4290.871} C_VEL
LIN {X 0,Y 530.992,Z 327.155,A -85,B 0,C 180,E1 -4293.257,E2 -4293.257} C_VEL
LIN {X 0,Y 531.003,Z 327.154,A -85,B 0,C 180,E1 -4295.953,E2 -4295.953} C_VEL
LIN {X 0,Y 530.991,Z 327.156,A -85,B 0,C 180,E1 -4299.063,E2 -4299.063} C_VEL
LIN {X 0,Y 531.003,Z 327.156,A -85,B 0,C 180,E1 -4302.278,E2 -4302.278} C_VEL
LIN {X 0,Y 531.006,Z 327.153,A -85,B 0,C 180,E1 -4305.436,E2 -4305.436} C_VEL
LIN {X 0,Y 531.036,Z 327.153,A -85,B 0,C 180,E1 -4308.551,E2 -4308.551} C_VEL
LIN {X 0,Y 531.049,Z 327.148,A -85,B 0,C 180,E1 -4311.63,E2 -4311.63} C_VEL
LIN {X 0,Y 531.113,Z 327.142,A -85,B 0,C 180,E1 -4314.686,E2 -4314.686} C_VEL
LIN {X 0,Y 531.133,Z 327.138,A -85,B 0,C 180,E1 -4317.726,E2 -4317.726} C_VEL
LIN {X 0,Y 531.147,Z 327.138,A -85,B 0,C 180,E1 -4320.759,E2 -4320.759} C_VEL
LIN {X 0,Y 531.099,Z 327.144,A -85,B 0,C 180,E1 -4323.035,E2 -4323.035} C_VEL
LIN {X 0,Y 531.074,Z 327.146,A -85,B 0,C 180,E1 -4326.078,E2 -4326.078} C_VEL
LIN {X 0,Y 531.021,Z 327.154,A -85,B 0,C 180,E1 -4329.139,E2 -4329.139} C_VEL
LIN {X 0,Y 531.032,Z 327.151,A -85,B 0,C 180,E1 -4332.226,E2 -4332.226} C_VEL
LIN {X 0,Y 530.987,Z 327.159,A -85,B 0,C 180,E1 -4335.351,E2 -4335.351} C_VEL
LIN {X 0,Y 531.007,Z 327.156,A -85,B 0,C 180,E1 -4337.723,E2 -4337.723} C_VEL
LIN {X 0,Y 530.991,Z 327.156,A -85,B 0,C 180,E1 -4340.939,E2 -4340.939} C_VEL
LIN {X 0,Y 530.971,Z 327.157,A -85,B 0,C 180,E1 -4344.225,E2 -4344.225} C_VEL
LIN {X 0,Y 531.004,Z 327.154,A -85,B 0,C 180,E1 -4346.744,E2 -4346.744} C_VEL
LIN {X 0,Y 530.993,Z 327.156,A -85,B 0,C 180,E1 -4349.322,E2 -4349.322} C_VEL
LIN {X 0,Y 530.962,Z 327.161,A -85,B 0,C 180,E1 -4352.102,E2 -4352.102} C_VEL
LIN {X 0,Y 530.984,Z 327.159,A -85,B 0,C 180,E1 -4354.856,E2 -4354.856} C_VEL
LIN {X 0,Y 530.96,Z 327.16,A -85,B 0,C 180,E1 -4357.509,E2 -4357.509} C_VEL
LIN {X 0,Y 530.977,Z 327.158,A -85,B 0,C 180,E1 -4360.434,E2 -4360.434} C_VEL
LIN {X 0,Y 530.964,Z 327.161,A -85,B 0,C 180,E1 -4363.283,E2 -4363.283} C_VEL
LIN {X 0,Y 530.982,Z 327.159,A -85,B 0,C 180,E1 -4365.622,E2 -4365.622} C_VEL
LIN {X 0,Y 530.995,Z 327.156,A -85,B 0,C 180,E1 -4368.566,E2 -4368.566} C_VEL
LIN {X 0,Y 530.955,Z 327.162,A -85,B 0,C 180,E1 -4371.531,E2 -4371.531} C_VEL
LIN {X 0,Y 530.984,Z 327.158,A -85,B 0,C 180,E1 -4374.384,E2 -4374.384} C_VEL
LIN {X 0,Y 531.055,Z 327.24,A -85,B 0,C 180,E1 -4375.432,E2 -4375.432} C_VEL
LIN {X 0,Y 531.693,Z 331.894,A -85,B 0,C 180,E1 -4377.185,E2 -4377.185} C_VEL
LIN {X 0,Y 531.583,Z 337.669,A -85,B 0,C 180,E1 -4379.245,E2 -4379.245} C_VEL
LIN {X 0,Y 531.328,Z 346.915,A -85,B 0,C 180,E1 -4382.424,E2 -4382.424} C_VEL
LIN {X 0,Y 531.157,Z 354.557,A -85,B 0,C 180,E1 -4384.951,E2 -4384.951} C_VEL
LIN {X 0,Y 531.002,Z 363.621,A -85,B 0,C 180,E1 -4387.892,E2 -4387.892} C_VEL
LIN {X 0,Y 530.841,Z 372.335,A -85,B 0,C 180,E1 -4390.673,E2 -4390.673} C_VEL
LIN {X 0,Y 530.762,Z 381.471,A -85,B 0,C 180,E1 -4393.461,E2 -4393.461} C_VEL
LIN {X 0,Y 530.664,Z 390.616,A -85,B 0,C 180,E1 -4396.21,E2 -4396.21} C_VEL
LIN {X 0,Y 530.604,Z 399.754,A -85,B 0,C 180,E1 -4398.937,E2 -4398.937} C_VEL
LIN {X 0,Y 530.605,Z 401.334,A -85,B 0,C 180,E1 -4399.339,E2 -4399.339} C_VEL
LIN {X 0,Y 531.546,Z 411.373,A -85,B 0,C 180,E1 -4399.623,E2 -4399.623} C_VEL
LIN {X 0,Y 531.421,Z 423.187,A -85,B 0,C 180,E1 -4400.101,E2 -4400.101} C_VEL
LIN {X 0,Y 531.236,Z 431.92,A -85,B 0,C 180,E1 -4400.578,E2 -4400.578} C_VEL
LIN {X 0,Y 531.101,Z 440.264,A -85,B 0,C 180,E1 -4401.152,E2 -4401.152} C_VEL
LIN {X 0,Y 530.946,Z 448.163,A -85,B 0,C 180,E1 -4401.82,E2 -4401.82} C_VEL
LIN {X 0,Y 530.789,Z 455.549,A -85,B 0,C 180,E1 -4402.584,E2 -4402.584} C_VEL
LIN {X 0,Y 530.701,Z 463.129,A -85,B 0,C 180,E1 -4403.549,E2 -4403.549} C_VEL
LIN {X 0,Y 530.596,Z 468.931,A -85,B 0,C 180,E1 -4404.49,E2 -4404.49} C_VEL
LIN {X 0,Y 530.506,Z 473.564,A -85,B 0,C 180,E1 -4405.442,E2 -4405.442} C_VEL
LIN {X 0,Y 530.525,Z 476.578,A -85,B 0,C 180,E1 -4406.203,E2 -4406.203} C_VEL
LIN {X 0,Y 530.469,Z 478.911,A -85,B 0,C 180,E1 -4406.963,E2 -4406.963} C_VEL
LIN {X 0,Y 530.412,Z 480.665,A -85,B 0,C 180,E1 -4407.723,E2 -4407.723} C_VEL
LIN {X 0,Y 530.36,Z 481.918,A -85,B 0,C 180,E1 -4408.482,E2 -4408.482} C_VEL
LIN {X 0,Y 530.34,Z 482.698,A -85,B 0,C 180,E1 -4409.242,E2 -4409.242} C_VEL
LIN {X 0,Y 530.34,Z 482.993,A -85,B 0,C 180,E1 -4410.001,E2 -4410.001} C_VEL
LIN {X 0,Y 530.34,Z 482.697,A -85,B 0,C 180,E1 -4410.76,E2 -4410.76} C_VEL
LIN {X 0,Y 530.36,Z 481.915,A -85,B 0,C 180,E1 -4411.52,E2 -4411.52} C_VEL
LIN {X 0,Y 530.412,Z 480.659,A -85,B 0,C 180,E1 -4412.279,E2 -4412.279} C_VEL
LIN {X 0,Y 530.493,Z 477.745,A -85,B 0,C 180,E1 -4413.419,E2 -4413.419} C_VEL
LIN {X 0,Y 530.544,Z 475.086,A -85,B 0,C 180,E1 -4414.179,E2 -4414.179} C_VEL
LIN {X 0,Y 530.542,Z 469.877,A -85,B 0,C 180,E1 -4415.321,E2 -4415.321} C_VEL
LIN {X 0,Y 530.729,Z 464.299,A -85,B 0,C 180,E1 -4416.271,E2 -4416.271} C_VEL
LIN {X 0,Y 530.774,Z 457.23,A -85,B 0,C 180,E1 -4417.227,E2 -4417.227} C_VEL
LIN {X 0,Y 530.919,Z 449.159,A -85,B 0,C 180,E1 -4418.086,E2 -4418.086} C_VEL
LIN {X 0,Y 531.087,Z 441.457,A -85,B 0,C 180,E1 -4418.754,E2 -4418.754} C_VEL
LIN {X 0,Y 531.199,Z 433.369,A -85,B 0,C 180,E1 -4419.328,E2 -4419.328} C_VEL
LIN {X 0,Y 531.354,Z 424.994,A -85,B 0,C 180,E1 -4419.806,E2 -4419.806} C_VEL
LIN {X 0,Y 531.469,Z 416.449,A -85,B 0,C 180,E1 -4420.188,E2 -4420.188} C_VEL
LIN {X 0,Y 531.469,Z 408.347,A -85,B 0,C 180,E1 -4420.465,E2 -4420.465} C_VEL
LIN {X 0,Y 530.57,Z 400.959,A -85,B 0,C 180,E1 -4420.688,E2 -4420.688} C_VEL
LIN {X 0,Y 530.666,Z 390.516,A -85,B 0,C 180,E1 -4423.792,E2 -4423.792} C_VEL
LIN {X 0,Y 530.732,Z 381.328,A -85,B 0,C 180,E1 -4426.542,E2 -4426.542} C_VEL
LIN {X 0,Y 530.844,Z 372.173,A -85,B 0,C 180,E1 -4429.329,E2 -4429.329} C_VEL
LIN {X 0,Y 530.972,Z 363.394,A -85,B 0,C 180,E1 -4432.1,E2 -4432.1} C_VEL
LIN {X 0,Y 531.184,Z 352.983,A -85,B 0,C 180,E1 -4435.468,E2 -4435.468} C_VEL
LIN {X 0,Y 531.352,Z 344.112,A -85,B 0,C 180,E1 -4438.436,E2 -4438.436} C_VEL
LIN {X 0,Y 531.613,Z 336.665,A -85,B 0,C 180,E1 -4441.037,E2 -4441.037} C_VEL
LIN {X 0,Y 531.676,Z 331.769,A -85,B 0,C 180,E1 -4442.818,E2 -4442.818} C_VEL
LIN {X 0,Y 530.989,Z 327.159,A -85,B 0,C 180,E1 -4444.691,E2 -4444.691} C_VEL
LIN {X 0,Y 530.971,Z 327.16,A -85,B 0,C 180,E1 -4447.508,E2 -4447.508} C_VEL
LIN {X 0,Y 530.986,Z 327.161,A -85,B 0,C 180,E1 -4450.433,E2 -4450.433} C_VEL
LIN {X 0,Y 530.97,Z 327.161,A -85,B 0,C 180,E1 -4453.495,E2 -4453.495} C_VEL
LIN {X 0,Y 530.96,Z 327.163,A -85,B 0,C 180,E1 -4456.505,E2 -4456.505} C_VEL
LIN {X 0,Y 530.99,Z 327.158,A -85,B 0,C 180,E1 -4458.977,E2 -4458.977} C_VEL
LIN {X 0,Y 530.96,Z 327.16,A -85,B 0,C 180,E1 -4461.529,E2 -4461.529} C_VEL
LIN {X 0,Y 530.96,Z 327.161,A -85,B 0,C 180,E1 -4464.38,E2 -4464.38} C_VEL
LIN {X 0,Y 530.972,Z 327.161,A -85,B 0,C 180,E1 -4467.133,E2 -4467.133} C_VEL
LIN {X 0,Y 530.966,Z 327.159,A -85,B 0,C 180,E1 -4469.802,E2 -4469.802} C_VEL
LIN {X 0,Y 531.017,Z 327.153,A -85,B 0,C 180,E1 -4472.468,E2 -4472.468} C_VEL
LIN {X 0,Y 531.011,Z 327.154,A -85,B 0,C 180,E1 -4474.942,E2 -4474.942} C_VEL
LIN {X 0,Y 530.978,Z 327.157,A -85,B 0,C 180,E1 -4478.246,E2 -4478.246} C_VEL
LIN {X 0,Y 530.998,Z 327.155,A -85,B 0,C 180,E1 -4480.677,E2 -4480.677} C_VEL
LIN {X 0,Y 530.976,Z 327.158,A -85,B 0,C 180,E1 -4483.07,E2 -4483.07} C_VEL
LIN {X 0,Y 531.023,Z 327.152,A -85,B 0,C 180,E1 -4485.435,E2 -4485.435} C_VEL
LIN {X 0,Y 531.043,Z 327.15,A -85,B 0,C 180,E1 -4488.549,E2 -4488.549} C_VEL
LIN {X 0,Y 531.041,Z 327.151,A -85,B 0,C 180,E1 -4491.629,E2 -4491.629} C_VEL
LIN {X 0,Y 531.123,Z 327.14,A -85,B 0,C 180,E1 -4494.685,E2 -4494.685} C_VEL
LIN {X 0,Y 531.14,Z 327.14,A -85,B 0,C 180,E1 -4497.724,E2 -4497.724} C_VEL
LIN {X 0,Y 531.158,Z 327.135,A -85,B 0,C 180,E1 -4500.757,E2 -4500.757} C_VEL
LIN {X 0,Y 531.107,Z 327.141,A -85,B 0,C 180,E1 -4503.033,E2 -4503.033} C_VEL
LIN {X 0,Y 531.087,Z 327.147,A -85,B 0,C 180,E1 -4506.076,E2 -4506.076} C_VEL
LIN {X 0,Y 531.017,Z 327.153,A -85,B 0,C 180,E1 -4509.138,E2 -4509.138} C_VEL
LIN {X 0,Y 531.044,Z 327.15,A -85,B 0,C 180,E1 -4512.224,E2 -4512.224} C_VEL
LIN {X 0,Y 530.998,Z 327.16,A -85,B 0,C 180,E1 -4515.349,E2 -4515.349} C_VEL
LIN {X 0,Y 530.943,Z 327.166,A -85,B 0,C 180,E1 -4517.724,E2 -4517.724} C_VEL
LIN {X 0,Y 530.807,Z 327.182,A -85,B 0,C 180,E1 -4518.527,E2 -4518.527} C_VEL
LIN {X 0,Y 530.76,Z 327.627,A -85,B 0,C 180,E1 -4519.331,E2 -4519.331} C_VEL
LIN {X 0,Y 530.703,Z 331.268,A -85,B 0,C 180,E1 -4522.027,E2 -4522.027} C_VEL
LIN {X 0,Y 530.649,Z 335.404,A -85,B 0,C 180,E1 -4525.074,E2 -4525.074} C_VEL
LIN {X 0,Y 530.573,Z 338.878,A -85,B 0,C 180,E1 -4527.619,E2 -4527.619} C_VEL
LIN {X 0,Y 530.538,Z 342.946,A -85,B 0,C 180,E1 -4530.564,E2 -4530.564} C_VEL
LIN {X 0,Y 530.46,Z 346.887,A -85,B 0,C 180,E1 -4533.417,E2 -4533.417} C_VEL
LIN {X 0,Y 530.42,Z 350.522,A -85,B 0,C 180,E1 -4536.075,E2 -4536.075} C_VEL
LIN {X 0,Y 530.413,Z 355.265,A -85,B 0,C 180,E1 -4539.431,E2 -4539.431} C_VEL
LIN {X 0,Y 531.59,Z 364.14,A -85,B 0,C 180,E1 -4539.731,E2 -4539.731} C_VEL
LIN {X 0,Y 531.424,Z 374.303,A -85,B 0,C 180,E1 -4540.16,E2 -4540.16} C_VEL
LIN {X 0,Y 531.345,Z 380.908,A -85,B 0,C 180,E1 -4540.51,E2 -4540.51} C_VEL
LIN {X 0,Y 530.669,Z 384.366,A -85,B 0,C 180,E1 -4540.712,E2 -4540.712} C_VEL
LIN {X 0,Y 527.714,Z 389.746,A -85,B 0,C 180,E1 -4541.024,E2 -4541.024} C_VEL
LIN {X 0,Y 524.718,Z 394.914,A -85,B 0,C 180,E1 -4541.376,E2 -4541.376} C_VEL
LIN {X 0,Y 523.984,Z 397.96,A -85,B 0,C 180,E1 -4541.642,E2 -4541.642} C_VEL
LIN {X 0,Y 523.863,Z 404.324,A -85,B 0,C 180,E1 -4542.284,E2 -4542.284} C_VEL
LIN {X 0,Y 523.715,Z 410.174,A -85,B 0,C 180,E1 -4542.987,E2 -4542.987} C_VEL
LIN {X 0,Y 523.582,Z 416.276,A -85,B 0,C 180,E1 -4543.88,E2 -4543.88} C_VEL
LIN {X 0,Y 523.54,Z 420.589,A -85,B 0,C 180,E1 -4544.644,E2 -4544.644} C_VEL
LIN {X 0,Y 523.416,Z 425.394,A -85,B 0,C 180,E1 -4545.715,E2 -4545.715} C_VEL
LIN {X 0,Y 523.376,Z 428.961,A -85,B 0,C 180,E1 -4546.776,E2 -4546.776} C_VEL
LIN {X 0,Y 523.341,Z 431.426,A -85,B 0,C 180,E1 -4547.82,E2 -4547.82} C_VEL
LIN {X 0,Y 523.309,Z 432.914,A -85,B 0,C 180,E1 -4548.847,E2 -4548.847} C_VEL
LIN {X 0,Y 523.258,Z 433.542,A -85,B 0,C 180,E1 -4549.957,E2 -4549.957} C_VEL
LIN {X 0,Y 523.276,Z 433.007,A -85,B 0,C 180,E1 -4551.166,E2 -4551.166} C_VEL
LIN {X 0,Y 523.267,Z 431.128,A -85,B 0,C 180,E1 -4552.411,E2 -4552.411} C_VEL
LIN {X 0,Y 523.379,Z 427.877,A -85,B 0,C 180,E1 -4553.674,E2 -4553.674} C_VEL
LIN {X 0,Y 523.469,Z 422.859,A -85,B 0,C 180,E1 -4554.98,E2 -4554.98} C_VEL
LIN {X 0,Y 523.566,Z 417.305,A -85,B 0,C 180,E1 -4556.035,E2 -4556.035} C_VEL
LIN {X 0,Y 523.673,Z 412.017,A -85,B 0,C 180,E1 -4556.845,E2 -4556.845} C_VEL
LIN {X 0,Y 523.795,Z 406.605,A -85,B 0,C 180,E1 -4557.54,E2 -4557.54} C_VEL
LIN {X 0,Y 523.917,Z 400.211,A -85,B 0,C 180,E1 -4558.229,E2 -4558.229} C_VEL
LIN {X 0,Y 524.077,Z 392.473,A -85,B 0,C 180,E1 -4558.916,E2 -4558.916} C_VEL
LIN {X 0,Y 524.221,Z 384.665,A -85,B 0,C 180,E1 -4559.484,E2 -4559.484} C_VEL
LIN {X 0,Y 524.407,Z 375.845,A -85,B 0,C 180,E1 -4559.996,E2 -4559.996} C_VEL
LIN {X 0,Y 524.555,Z 366.781,A -85,B 0,C 180,E1 -4560.402,E2 -4560.402} C_VEL
LIN {X 0,Y 524.231,Z 361.357,A -85,B 0,C 180,E1 -4560.603,E2 -4560.603} C_VEL
LIN {X 0,Y 523.379,Z 355.541,A -85,B 0,C 180,E1 -4560.811,E2 -4560.811} C_VEL
LIN {X 0,Y 523.43,Z 350.866,A -85,B 0,C 180,E1 -4564.102,E2 -4564.102} C_VEL
LIN {X 0,Y 523.397,Z 346.661,A -85,B 0,C 180,E1 -4567.082,E2 -4567.082} C_VEL
LIN {X 0,Y 523.447,Z 342.068,A -85,B 0,C 180,E1 -4570.387,E2 -4570.387} C_VEL
LIN {X 0,Y 523.506,Z 338.696,A -85,B 0,C 180,E1 -4572.821,E2 -4572.821} C_VEL
LIN {X 0,Y 523.527,Z 334.352,A -85,B 0,C 180,E1 -4576.016,E2 -4576.016} C_VEL
LIN {X 0,Y 523.71,Z 330.045,A -85,B 0,C 180,E1 -4579.17,E2 -4579.17} C_VEL
LIN {X 0,Y 523.683,Z 328.07,A -85,B 0,C 180,E1 -4580.732,E2 -4580.732} C_VEL
LIN {X 0,Y 524.02,Z 328.024,A -85,B 0,C 180,E1 -4583.066,E2 -4583.066} C_VEL
LIN {X 0,Y 523.96,Z 328.031,A -85,B 0,C 180,E1 -4585.383,E2 -4585.383} C_VEL
LIN {X 0,Y 524.1,Z 328.014,A -85,B 0,C 180,E1 -4587.693,E2 -4587.693} C_VEL
LIN {X 0,Y 524.115,Z 328.014,A -85,B 0,C 180,E1 -4590.767,E2 -4590.767} C_VEL
LIN {X 0,Y 524.065,Z 328.02,A -85,B 0,C 180,E1 -4593.074,E2 -4593.074} C_VEL
LIN {X 0,Y 524.037,Z 328.023,A -85,B 0,C 180,E1 -4596.158,E2 -4596.158} C_VEL
LIN {X 0,Y 523.994,Z 328.029,A -85,B 0,C 180,E1 -4599.261,E2 -4599.261} C_VEL
LIN {X 0,Y 524.012,Z 328.028,A -85,B 0,C 180,E1 -4601.75,E2 -4601.75} C_VEL
LIN {X 0,Y 523.979,Z 328.029,A -85,B 0,C 180,E1 -4605.052,E2 -4605.052} C_VEL
LIN {X 0,Y 523.951,Z 328.034,A -85,B 0,C 180,E1 -4607.968,E2 -4607.968} C_VEL
LIN {X 0,Y 523.959,Z 328.033,A -85,B 0,C 180,E1 -4610.409,E2 -4610.409} C_VEL
LIN {X 0,Y 523.903,Z 328.041,A -85,B 0,C 180,E1 -4612.893,E2 -4612.893} C_VEL
LIN {X 0,Y 523.941,Z 328.035,A -85,B 0,C 180,E1 -4615.418,E2 -4615.418} C_VEL
LIN {X 0,Y 523.957,Z 328.032,A -85,B 0,C 180,E1 -4617.998,E2 -4617.998} C_VEL
LIN {X 0,Y 523.938,Z 328.034,A -85,B 0,C 180,E1 -4620.856,E2 -4620.856} C_VEL
LIN {X 0,Y 523.948,Z 328.034,A -85,B 0,C 180,E1 -4623.735,E2 -4623.735} C_VEL
LIN {X 0,Y 523.911,Z 328.038,A -85,B 0,C 180,E1 -4626.405,E2 -4626.405} C_VEL
LIN {X 0,Y 523.945,Z 328.034,A -85,B 0,C 180,E1 -4629.081,E2 -4629.081} C_VEL
LIN {X 0,Y 523.951,Z 328.034,A -85,B 0,C 180,E1 -4632.117,E2 -4632.117} C_VEL
LIN {X 0,Y 523.941,Z 328.035,A -85,B 0,C 180,E1 -4635.309,E2 -4635.309} C_VEL
LIN {X 0,Y 523.957,Z 328.032,A -85,B 0,C 180,E1 -4638.688,E2 -4638.688} C_VEL
LIN {X 0,Y 523.939,Z 328.035,A -85,B 0,C 180,E1 -4641.075,E2 -4641.075} C_VEL
LIN {X 0,Y 523.915,Z 328.037,A -85,B 0,C 180,E1 -4643.828,E2 -4643.828} C_VEL
LIN {X 0,Y 523.93,Z 328.038,A -85,B 0,C 180,E1 -4646.636,E2 -4646.636} C_VEL
LIN {X 0,Y 523.949,Z 328.033,A -85,B 0,C 180,E1 -4649.357,E2 -4649.357} C_VEL
LIN {X 0,Y 523.965,Z 328.031,A -85,B 0,C 180,E1 -4652.281,E2 -4652.281} C_VEL
LIN {X 0,Y 523.94,Z 328.035,A -85,B 0,C 180,E1 -4654.582,E2 -4654.582} C_VEL
LIN {X 0,Y 523.937,Z 328.035,A -85,B 0,C 180,E1 -4657.109,E2 -4657.109} C_VEL
LIN {X 0,Y 523.965,Z 328.032,A -85,B 0,C 180,E1 -4659.866,E2 -4659.866} C_VEL
LIN {X 0,Y 523.958,Z 328.032,A -85,B 0,C 180,E1 -4662.838,E2 -4662.838} C_VEL
LIN {X 0,Y 523.963,Z 328.031,A -85,B 0,C 180,E1 -4665.236,E2 -4665.236} C_VEL
LIN {X 0,Y 524.002,Z 328.029,A -85,B 0,C 180,E1 -4668.395,E2 -4668.395} C_VEL
LIN {X 0,Y 523.996,Z 328.027,A -85,B 0,C 180,E1 -4671.517,E2 -4671.517} C_VEL
LIN {X 0,Y 524.074,Z 328.019,A -85,B 0,C 180,E1 -4674.614,E2 -4674.614} C_VEL
LIN {X 0,Y 524.104,Z 328.014,A -85,B 0,C 180,E1 -4677.695,E2 -4677.695} C_VEL
LIN {X 0,Y 524.117,Z 328.013,A -85,B 0,C 180,E1 -4680.769,E2 -4680.769} C_VEL
LIN {X 0,Y 524.066,Z 328.02,A -85,B 0,C 180,E1 -4683.076,E2 -4683.076} C_VEL
LIN {X 0,Y 524.036,Z 328.022,A -85,B 0,C 180,E1 -4686.16,E2 -4686.16} C_VEL
LIN {X 0,Y 523.99,Z 328.031,A -85,B 0,C 180,E1 -4689.263,E2 -4689.263} C_VEL
LIN {X 0,Y 524.014,Z 328.027,A -85,B 0,C 180,E1 -4691.752,E2 -4691.752} C_VEL
LIN {X 0,Y 523.983,Z 328.029,A -85,B 0,C 180,E1 -4695.053,E2 -4695.053} C_VEL
LIN {X 0,Y 523.955,Z 328.033,A -85,B 0,C 180,E1 -4697.97,E2 -4697.97} C_VEL
LIN {X 0,Y 523.963,Z 328.032,A -85,B 0,C 180,E1 -4700.411,E2 -4700.411} C_VEL
LIN {X 0,Y 523.908,Z 328.039,A -85,B 0,C 180,E1 -4702.894,E2 -4702.894} C_VEL
LIN {X 0,Y 523.946,Z 328.034,A -85,B 0,C 180,E1 -4705.42,E2 -4705.42} C_VEL
LIN {X 0,Y 523.963,Z 328.031,A -85,B 0,C 180,E1 -4708,E2 -4708} C_VEL
LIN {X 0,Y 523.942,Z 328.035,A -85,B 0,C 180,E1 -4710.857,E2 -4710.857} C_VEL
LIN {X 0,Y 523.956,Z 328.032,A -85,B 0,C 180,E1 -4713.736,E2 -4713.736} C_VEL
LIN {X 0,Y 523.916,Z 328.037,A -85,B 0,C 180,E1 -4716.405,E2 -4716.405} C_VEL
LIN {X 0,Y 523.916,Z 328.038,A -85,B 0,C 180,E1 -4719.086,E2 -4719.086} C_VEL
LIN {X 0,Y 523.951,Z 328.035,A -85,B 0,C 180,E1 -4722.119,E2 -4722.119} C_VEL
LIN {X 0,Y 523.95,Z 328.034,A -85,B 0,C 180,E1 -4725.31,E2 -4725.31} C_VEL
LIN {X 0,Y 523.956,Z 328.033,A -85,B 0,C 180,E1 -4728.69,E2 -4728.69} C_VEL
LIN {X 0,Y 523.912,Z 328.038,A -85,B 0,C 180,E1 -4731.9,E2 -4731.9} C_VEL
LIN {X 0,Y 524.014,Z 328.107,A -85,B 0,C 180,E1 -4735.251,E2 -4735.251} C_VEL
LIN {X 0,Y 524.704,Z 333.072,A -85,B 0,C 180,E1 -4737.15,E2 -4737.15} C_VEL
LIN {X 0,Y 524.552,Z 339.289,A -85,B 0,C 180,E1 -4739.396,E2 -4739.396} C_VEL
LIN {X 0,Y 524.326,Z 347.347,A -85,B 0,C 180,E1 -4742.209,E2 -4742.209} C_VEL
LIN {X 0,Y 524.1,Z 355.662,A -85,B 0,C 180,E1 -4745.015,E2 -4745.015} C_VEL
LIN {X 0,Y 523.941,Z 363.985,A -85,B 0,C 180,E1 -4747.751,E2 -4747.751} C_VEL
LIN {X 0,Y 523.782,Z 373.438,A -85,B 0,C 180,E1 -4750.809,E2 -4750.809} C_VEL
LIN {X 0,Y 523.662,Z 382.551,A -85,B 0,C 180,E1 -4753.631,E2 -4753.631} C_VEL
LIN {X 0,Y 523.562,Z 391.693,A -85,B 0,C 180,E1 -4756.415,E2 -4756.415} C_VEL
LIN {X 0,Y 523.492,Z 400.964,A -85,B 0,C 180,E1 -4759.192,E2 -4759.192} C_VEL
LIN {X 0,Y 524.558,Z 411.015,A -85,B 0,C 180,E1 -4759.483,E2 -4759.483} C_VEL
LIN {X 0,Y 524.399,Z 422.839,A -85,B 0,C 180,E1 -4759.967,E2 -4759.967} C_VEL
LIN {X 0,Y 524.201,Z 431.574,A -85,B 0,C 180,E1 -4760.451,E2 -4760.451} C_VEL
LIN {X 0,Y 524.062,Z 439.921,A -85,B 0,C 180,E1 -4761.032,E2 -4761.032} C_VEL
LIN {X 0,Y 523.899,Z 447.822,A -85,B 0,C 180,E1 -4761.71,E2 -4761.71} C_VEL
LIN {X 0,Y 523.72,Z 455.21,A -85,B 0,C 180,E1 -4762.483,E2 -4762.483} C_VEL
LIN {X 0,Y 523.609,Z 461.884,A -85,B 0,C 180,E1 -4763.337,E2 -4763.337} C_VEL
LIN {X 0,Y 523.52,Z 468.597,A -85,B 0,C 180,E1 -4764.416,E2 -4764.416} C_VEL
LIN {X 0,Y 523.406,Z 473.231,A -85,B 0,C 180,E1 -4765.38,E2 -4765.38} C_VEL
LIN {X 0,Y 523.454,Z 476.247,A -85,B 0,C 180,E1 -4766.152,E2 -4766.152} C_VEL
LIN {X 0,Y 523.379,Z 478.58,A -85,B 0,C 180,E1 -4766.922,E2 -4766.922} C_VEL
LIN {X 0,Y 523.336,Z 480.335,A -85,B 0,C 180,E1 -4767.692,E2 -4767.692} C_VEL
LIN {X 0,Y 523.273,Z 481.591,A -85,B 0,C 180,E1 -4768.462,E2 -4768.462} C_VEL
LIN {X 0,Y 523.248,Z 482.373,A -85,B 0,C 180,E1 -4769.231,E2 -4769.231} C_VEL
LIN {X 0,Y 523.248,Z 482.668,A -85,B 0,C 180,E1 -4770.001,E2 -4770.001} C_VEL
LIN {X 0,Y 523.248,Z 482.371,A -85,B 0,C 180,E1 -4770.771,E2 -4770.771} C_VEL
LIN {X 0,Y 523.273,Z 481.585,A -85,B 0,C 180,E1 -4771.54,E2 -4771.54} C_VEL
LIN {X 0,Y 523.336,Z 480.324,A -85,B 0,C 180,E1 -4772.31,E2 -4772.31} C_VEL
LIN {X 0,Y 523.405,Z 477.405,A -85,B 0,C 180,E1 -4773.465,E2 -4773.465} C_VEL
LIN {X 0,Y 523.45,Z 474.742,A -85,B 0,C 180,E1 -4774.236,E2 -4774.236} C_VEL
LIN {X 0,Y 523.485,Z 469.531,A -85,B 0,C 180,E1 -4775.393,E2 -4775.393} C_VEL
LIN {X 0,Y 523.614,Z 463.389,A -85,B 0,C 180,E1 -4776.445,E2 -4776.445} C_VEL
LIN {X 0,Y 523.703,Z 456.869,A -85,B 0,C 180,E1 -4777.325,E2 -4777.325} C_VEL
LIN {X 0,Y 523.852,Z 448.792,A -85,B 0,C 180,E1 -4778.196,E2 -4778.196} C_VEL
LIN {X 0,Y 524.042,Z 441.086,A -85,B 0,C 180,E1 -4778.873,E2 -4778.873} C_VEL
LIN {X 0,Y 524.17,Z 432.993,A -85,B 0,C 180,E1 -4779.454,E2 -4779.454} C_VEL
LIN {X 0,Y 524.347,Z 424.612,A -85,B 0,C 180,E1 -4779.938,E2 -4779.938} C_VEL
LIN {X 0,Y 524.501,Z 416.063,A -85,B 0,C 180,E1 -4780.325,E2 -4780.325} C_VEL
LIN {X 0,Y 524.37,Z 408.364,A -85,B 0,C 180,E1 -4780.596,E2 -4780.596} C_VEL
LIN {X 0,Y 523.495,Z 400.616,A -85,B 0,C 180,E1 -4780.834,E2 -4780.834} C_VEL
LIN {X 0,Y 523.562,Z 391.552,A -85,B 0,C 180,E1 -4783.587,E2 -4783.587} C_VEL
LIN {X 0,Y 523.659,Z 383.684,A -85,B 0,C 180,E1 -4785.971,E2 -4785.971} C_VEL
LIN {X 0,Y 523.771,Z 374.522,A -85,B 0,C 180,E1 -4788.787,E2 -4788.787} C_VEL
LIN {X 0,Y 523.903,Z 365.551,A -85,B 0,C 180,E1 -4791.649,E2 -4791.649} C_VEL
LIN {X 0,Y 524.091,Z 355.336,A -85,B 0,C 180,E1 -4794.988,E2 -4794.988} C_VEL
LIN {X 0,Y 524.31,Z 346.499,A -85,B 0,C 180,E1 -4797.98,E2 -4797.98} C_VEL
LIN {X 0,Y 524.552,Z 339.053,A -85,B 0,C 180,E1 -4800.607,E2 -4800.607} C_VEL
LIN {X 0,Y 524.706,Z 332.949,A -85,B 0,C 180,E1 -4802.852,E2 -4802.852} C_VEL
LIN {X 0,Y 523.96,Z 328.035,A -85,B 0,C 180,E1 -4804.838,E2 -4804.838} C_VEL
LIN {X 0,Y 523.92,Z 328.04,A -85,B 0,C 180,E1 -4808.102,E2 -4808.102} C_VEL
LIN {X 0,Y 523.944,Z 328.037,A -85,B 0,C 180,E1 -4811.093,E2 -4811.093} C_VEL
LIN {X 0,Y 523.941,Z 328.038,A -85,B 0,C 180,E1 -4814.229,E2 -4814.229} C_VEL
LIN {X 0,Y 523.922,Z 328.037,A -85,B 0,C 180,E1 -4816.833,E2 -4816.833} C_VEL
LIN {X 0,Y 523.945,Z 328.036,A -85,B 0,C 180,E1 -4818.908,E2 -4818.908} C_VEL
LIN {X 0,Y 523.92,Z 328.037,A -85,B 0,C 180,E1 -4821.898,E2 -4821.898} C_VEL
LIN {X 0,Y 523.93,Z 328.037,A -85,B 0,C 180,E1 -4824.911,E2 -4824.911} C_VEL
LIN {X 0,Y 523.941,Z 328.034,A -85,B 0,C 180,E1 -4827.68,E2 -4827.68} C_VEL
LIN {X 0,Y 523.959,Z 328.034,A -85,B 0,C 180,E1 -4830.677,E2 -4830.677} C_VEL
LIN {X 0,Y 523.98,Z 328.03,A -85,B 0,C 180,E1 -4833.728,E2 -4833.728} C_VEL
LIN {X 0,Y 523.932,Z 328.037,A -85,B 0,C 180,E1 -4836.27,E2 -4836.27} C_VEL
LIN {X 0,Y 523.952,Z 328.035,A -85,B 0,C 180,E1 -4838.766,E2 -4838.766} C_VEL
LIN {X 0,Y 523.953,Z 328.035,A -85,B 0,C 180,E1 -4841.22,E2 -4841.22} C_VEL
LIN {X 0,Y 523.934,Z 328.037,A -85,B 0,C 180,E1 -4843.638,E2 -4843.638} C_VEL
LIN {X 0,Y 523.942,Z 328.036,A -85,B 0,C 180,E1 -4846.027,E2 -4846.027} C_VEL
LIN {X 0,Y 524.019,Z 328.026,A -85,B 0,C 180,E1 -4848.394,E2 -4848.394} C_VEL
LIN {X 0,Y 523.993,Z 328.029,A -85,B 0,C 180,E1 -4851.515,E2 -4851.515} C_VEL
LIN {X 0,Y 524.083,Z 328.017,A -85,B 0,C 180,E1 -4854.613,E2 -4854.613} C_VEL
LIN {X 0,Y 524.113,Z 328.016,A -85,B 0,C 180,E1 -4857.694,E2 -4857.694} C_VEL
LIN {X 0,Y 524.128,Z 328.011,A -85,B 0,C 180,E1 -4860.768,E2 -4860.768} C_VEL
LIN {X 0,Y 524.073,Z 328.017,A -85,B 0,C 180,E1 -4863.074,E2 -4863.074} C_VEL
LIN {X 0,Y 524.049,Z 328.023,A -85,B 0,C 180,E1 -4866.158,E2 -4866.158} C_VEL
LIN {X 0,Y 523.988,Z 328.03,A -85,B 0,C 180,E1 -4869.261,E2 -4869.261} C_VEL
LIN {X 0,Y 524.007,Z 328.028,A -85,B 0,C 180,E1 -4871.738,E2 -4871.738} C_VEL
LIN {X 0,Y 523.996,Z 328.029,A -85,B 0,C 180,E1 -4875.051,E2 -4875.051} C_VEL
LIN {X 0,Y 523.854,Z 328.049,A -85,B 0,C 180,E1 -4877.972,E2 -4877.972} C_VEL
LIN {X 0,Y 523.72,Z 328.065,A -85,B 0,C 180,E1 -4878.787,E2 -4878.787} C_VEL
LIN {X 0,Y 523.705,Z 329.344,A -85,B 0,C 180,E1 -4880.05,E2 -4880.05} C_VEL
LIN {X 0,Y 523.591,Z 333.163,A -85,B 0,C 180,E1 -4882.907,E2 -4882.907} C_VEL
LIN {X 0,Y 523.585,Z 336.571,A -85,B 0,C 180,E1 -4885.437,E2 -4885.437} C_VEL
LIN {X 0,Y 523.5,Z 340.063,A -85,B 0,C 180,E1 -4888.025,E2 -4888.025} C_VEL
LIN {X 0,Y 523.461,Z 343.838,A -85,B 0,C 180,E1 -4890.765,E2 -4890.765} C_VEL
LIN {X 0,Y 523.388,Z 347.774,A -85,B 0,C 180,E1 -4893.64,E2 -4893.64} C_VEL
LIN {X 0,Y 523.326,Z 351.393,A -85,B 0,C 180,E1 -4896.314,E2 -4896.314} C_VEL
LIN {X 0,Y 523.328,Z 355.63,A -85,B 0,C 180,E1 -4899.291,E2 -4899.291} C_VEL
LIN {X 0,Y 524.608,Z 365.719,A -85,B 0,C 180,E1 -4899.643,E2 -4899.643} C_VEL
LIN {X 0,Y 524.435,Z 374.738,A -85,B 0,C 180,E1 -4900.033,E2 -4900.033} C_VEL
LIN {X 0,Y 524.323,Z 382.668,A -85,B 0,C 180,E1 -4900.474,E2 -4900.474} C_VEL
LIN {X 0,Y 524.095,Z 391.302,A -85,B 0,C 180,E1 -4901.076,E2 -4901.076} C_VEL
LIN {X 0,Y 523.984,Z 397.96,A -85,B 0,C 180,E1 -4901.642,E2 -4901.642} C_VEL
LIN {X 0,Y 523.266,Z 402.472,A -85,B 0,C 180,E1 -4902.063,E2 -4902.063} C_VEL
LIN {X 0,Y 520.203,Z 409.314,A -85,B 0,C 180,E1 -4902.798,E2 -4902.798} C_VEL
LIN {X 0,Y 517.191,Z 415.338,A -85,B 0,C 180,E1 -4903.595,E2 -4903.595} C_VEL
LIN {X 0,Y 516.499,Z 418.569,A -85,B 0,C 180,E1 -4904.126,E2 -4904.126} C_VEL
LIN {X 0,Y 516.411,Z 424.332,A -85,B 0,C 180,E1 -4905.294,E2 -4905.294} C_VEL
LIN {X 0,Y 516.34,Z 427.64,A -85,B 0,C 180,E1 -4906.168,E2 -4906.168} C_VEL
LIN {X 0,Y 516.279,Z 430.783,A -85,B 0,C 180,E1 -4907.313,E2 -4907.313} C_VEL
LIN {X 0,Y 516.231,Z 432.823,A -85,B 0,C 180,E1 -4908.482,E2 -4908.482} C_VEL
